# B&R Automation Studio project RS15_RX_30005_r00 (part 6)

### Program Logical/BagMachine_Section/EnvBag/Axis12/A12_Cycle (IEC) - A new program

#### A12_CycleInit.st - Initialization code
```iecst
(********************************************************************
 * COPYRIGHT -- .
 ********************************************************************
 * Program: A12_Cycle
 * File: A12_CycleInit.st
 * Author: dominique
 * Created: November 21, 2011
 ********************************************************************
 * Implementation of program A12_Cycle
 ********************************************************************)

PROGRAM _INIT

  gstCycA[12].CycManTimSet.uiMasterParID := 428 ; // ParID 428 = CTRL Position controller: Input set position (in case real axis)

END_PROGRAM
```

#### A12_Cycle.var - Local variables
```iecst
(********************************************************************
 * COPYRIGHT -- .
 ********************************************************************
 * Program: A12_Cycle
 * File: A12_Cycle.var
 * Author: dominique
 * Created: November 21, 2011
 ********************************************************************
 * Local variables of program A12_Cycle
 ********************************************************************)

VAR
  iTest_          : ARRAY [0..15] OF INT ;
  rTempActPhasDeg : ARRAY[0..15] OF REAL ;
  rTempActOffsetInch : ARRAY[0..15] OF REAL ;
  rTemp_          : ARRAY[0..15] OF REAL ;
  stTON_01        : TON ;
END_VAR

VAR CONSTANT

END_VAR
```

### Program Logical/BagMachine_Section/EnvBag/Axis12/A12_Ref_V1 (IEC) - Reference Routine

#### A12_RefCyclic.ld - Cyclic code
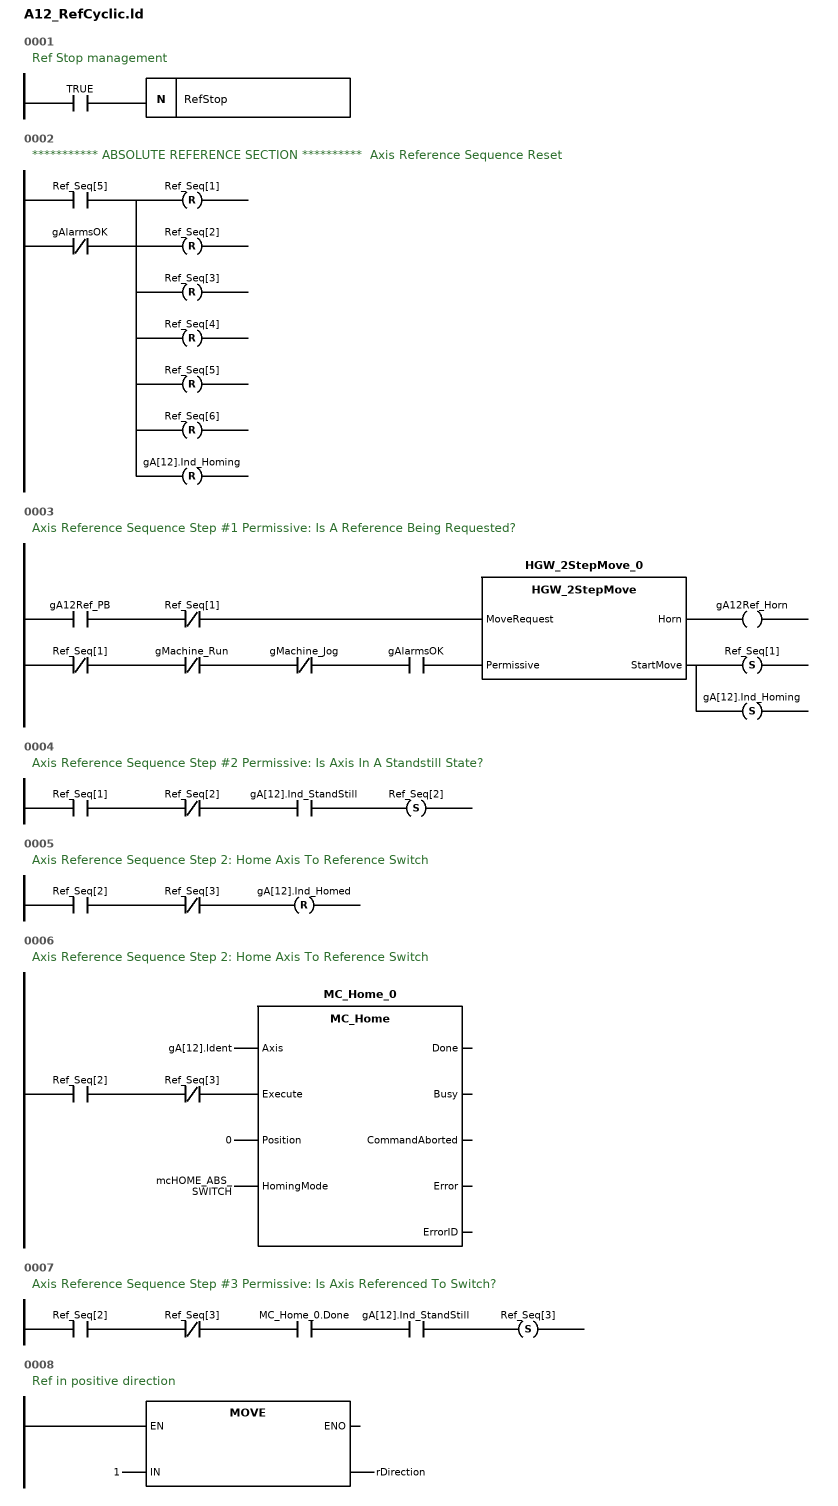
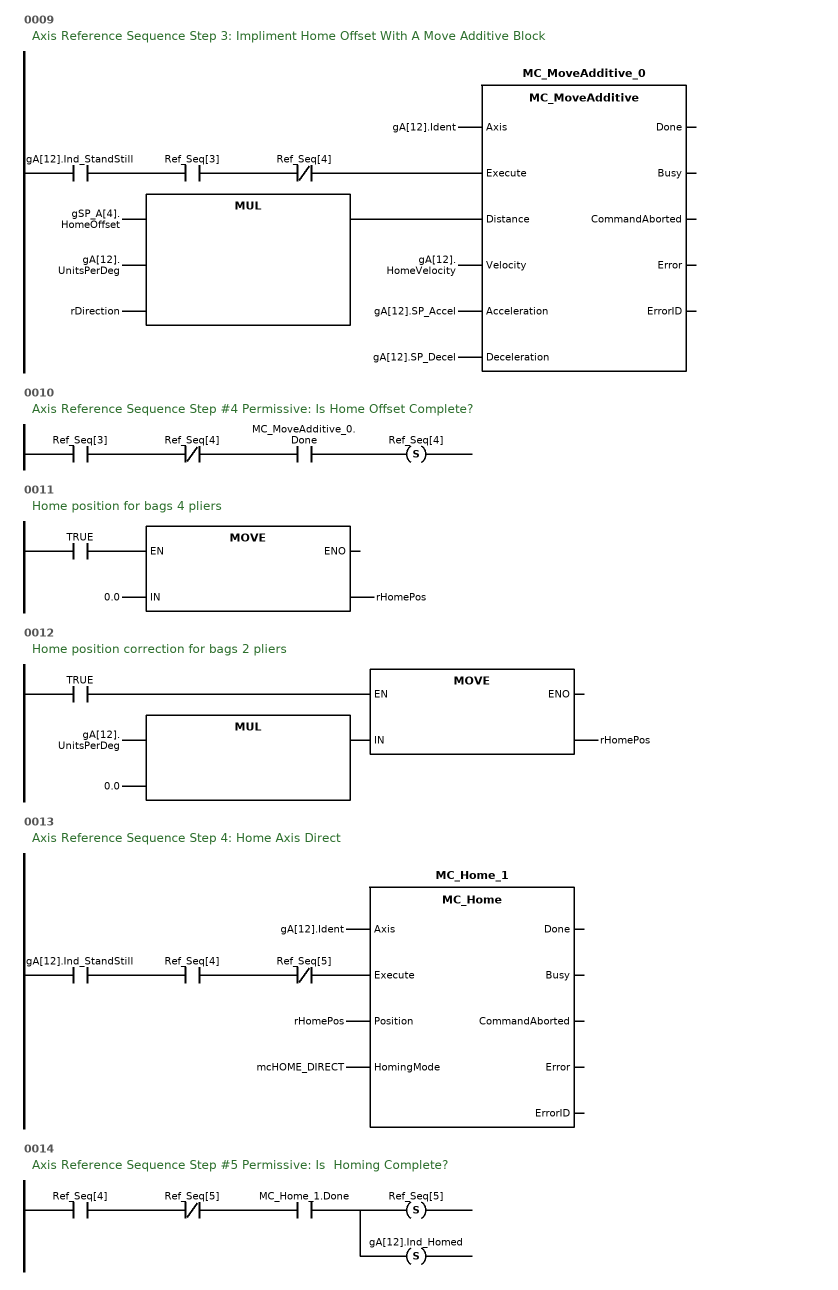
Ladder, written as Structured Text:
```iecst
(********************************************************************
 * COPYRIGHT -- Microsoft
 ********************************************************************
 * Program: A4_Ref
 * File: A4_RefCyclic.ld
 * Author: pkiel
 * Created: July 19, 2011
 ********************************************************************
 * Implementation of program A4_Ref
 ********************************************************************)

PROGRAM _CYCLIC
VAR
    _p1 : BOOL;
    _p2 : BOOL;
END_VAR
(* Network 1: Ref Stop management *)
RefStop;

(* Network 2: *********** ABSOLUTE REFERENCE SECTION **********  Axis Reference Sequence Reset *)
_p1 := Ref_Seq[5];
IF Ref_Seq[5] OR NOT gAlarmsOK THEN Ref_Seq[1] := FALSE; END_IF;
IF _p1 OR NOT gAlarmsOK THEN
    Ref_Seq[2] := FALSE;
    Ref_Seq[3] := FALSE;
    Ref_Seq[4] := FALSE;
    Ref_Seq[5] := FALSE;
    Ref_Seq[6] := FALSE;
    gA[12].Ind_Homing := FALSE;
END_IF;

(* Network 3: Axis Reference Sequence Step #1 Permissive: Is A Reference Being Requested? *)
HGW_2StepMove_0(MoveRequest := gA12Ref_PB AND NOT Ref_Seq[1], Permissive := NOT Ref_Seq[1] AND NOT gMachine_Run AND NOT gMachine_Jog AND gAlarmsOK);
gA12Ref_Horn := HGW_2StepMove_0.Horn;
IF HGW_2StepMove_0.StartMove THEN
    Ref_Seq[1] := TRUE;
    gA[12].Ind_Homing := TRUE;
END_IF;

(* Network 4: Axis Reference Sequence Step #2 Permissive: Is Axis In A Standstill State? *)
IF Ref_Seq[1] AND NOT Ref_Seq[2] AND gA[12].Ind_StandStill THEN Ref_Seq[2] := TRUE; END_IF;

(* Network 5: Axis Reference Sequence Step 2: Home Axis To Reference Switch *)
IF Ref_Seq[2] AND NOT Ref_Seq[3] THEN gA[12].Ind_Homed := FALSE; END_IF;

(* Network 6: Axis Reference Sequence Step 2: Home Axis To Reference Switch *)
MC_Home_0(Axis := gA[12].Ident, Execute := Ref_Seq[2] AND NOT Ref_Seq[3], Position := 0, HomingMode := mcHOME_ABS_SWITCH);

(* Network 7: Axis Reference Sequence Step #3 Permissive: Is Axis Referenced To Switch? *)
IF Ref_Seq[2] AND NOT Ref_Seq[3] AND MC_Home_0.Done AND gA[12].Ind_StandStill THEN
    Ref_Seq[3] := TRUE;
END_IF;

(* Network 8: Ref in positive direction  *)
rDirection := 1;

(* Network 9: Axis Reference Sequence Step 3: Impliment Home Offset With A Move Additive Block *)
MC_MoveAdditive_0(Axis := gA[12].Ident, Execute := gA[12].Ind_StandStill AND Ref_Seq[3] AND NOT Ref_Seq[4], Distance := gSP_A[4].HomeOffset * gA[12].UnitsPerDeg * rDirection, Velocity := gA[12].HomeVelocity, Acceleration := gA[12].SP_Accel, Deceleration := gA[12].SP_Decel);

(* Network 10: Axis Reference Sequence Step #4 Permissive: Is Home Offset Complete? *)
IF Ref_Seq[3] AND NOT Ref_Seq[4] AND MC_MoveAdditive_0.Done THEN Ref_Seq[4] := TRUE; END_IF;

(* Network 11: Home position for bags 4 pliers  *)
rHomePos := 0.0;

(* Network 12: Home position correction for bags 2 pliers *)
rHomePos := gA[12].UnitsPerDeg * 0.0;

(* Network 13: Axis Reference Sequence Step 4: Home Axis Direct *)
MC_Home_1(Axis := gA[12].Ident, Execute := gA[12].Ind_StandStill AND Ref_Seq[4] AND NOT Ref_Seq[5], Position := rHomePos, HomingMode := mcHOME_DIRECT);

(* Network 14: Axis Reference Sequence Step #5 Permissive: Is  Homing Complete? *)
_p2 := Ref_Seq[4] AND NOT Ref_Seq[5] AND MC_Home_1.Done;
IF Ref_Seq[4] AND NOT Ref_Seq[5] AND MC_Home_1.Done THEN Ref_Seq[5] := TRUE; END_IF;
IF _p2 THEN gA[12].Ind_Homed := TRUE; END_IF;
END_PROGRAM
```

### Package Logical/BagMachine_Section/EnvBag/Axis13 - Tearing Envelope Bag Axis     TearEB  Axis

### Program Logical/BagMachine_Section/EnvBag/Axis13/A13_Automat

#### A13_Automat.var
```iecst
(********************************************************************
 * COPYRIGHT -- Microsoft
 ********************************************************************
 * Program: A13_Automat
 * File: A13_Automat.var
 * Author: dominique
 * Created: November 21, 2011
 ********************************************************************
 * Local variables of program A13_Automat
 ********************************************************************)
VAR
	AutData : MC_AUTDATA_TYP;
	AutomatStart : BOOL;
	ErrorID : UINT;
	MasterOffset : REAL;
  MasterParID : UINT;
  uiMasterParID1 : UINT;
  uiSP_MasterParID : UINT;
  uiiSP_Master : UDINT;
  bCmdSynchroOn : BOOL ;
  bCmdSynchroOff : BOOL ;
  bCmdSynchroOn1 : BOOL ;
  bCmdSynchroOff1 : BOOL ;
  uiiSP_MasterFactor : UDINT ;
  uiiSP_SlaveFactor : UDINT ;
	MC_BR_AutControl_0 : MC_BR_AutControl;
  uiMC_BR_AutControl_0_MemoErrorID : UINT ;
  MC_BR_InitMasterParIDTransfer_0 : MC_BR_InitMasterParIDTransfer;
  MC_BR_InitMasterParIDTransfer_1 : MC_BR_InitMasterParIDTransfer;
  ParID_Ready : BOOL;
  ParID_Ready1 : BOOL;
	PositionMOD : DINT;
	PositionOffset : DINT;
	SlaveStartOffset : REAL;
	Synch_Request : BOOL;
  bTest_ : ARRAY[0..9] OF  BOOL;
  iTest_ : ARRAY[0..9] OF  INT;
  rTest_ : ARRAY[0..9] OF  REAL;
  rMaCompDist : REAL ;
  rSPMaPos    : REAL ;
  rOffsetDeg  : REAL ;
  rSlCompDist : REAL ;
  rTemp_      : ARRAY[0..9] OF REAL ;
  usiMemoStat : USINT;
  iIndex : INT ;
  rMaCompDistStat6 : REAL;
  rSlCompDistStat6 : REAL;
  rMasterFactor5 : REAL;
  iiMasterFactor5 : DINT;
  iiSlaveFactor5  : DINT;
  rSlave_AxisPeriod : REAL ;
  rSlave_TimingAxisPeriod : REAL ;
  MC_BR_InitAutState_0 : MC_BR_InitAutState;
  uiInitAutState_0_MemoErrorID : UINT ;
END_VAR
```

#### A13_AutomatCyclic.st
```iecst
(********************************************************************
 * COPYRIGHT -- Microsoft
 ********************************************************************
 * Program: A13_Automat
 * File: A13_AutomatCyclic.st
 * Author: dominique
 * Created: November 21, 2011
 ********************************************************************
 * Implementation of program A13_Automat
 ********************************************************************)

PROGRAM _CYCLIC

    // Synchro ratio Master/Slave
    iIndex := MC_BR_AutControl_0.ActualStateIndex ;
    IF gRecipeActive.bSelEnvBProd THEN
      CASE iIndex OF
        3 : // Master = EnvB Axis
           //gA[13].rRSynNum := 4.0 ;       D.M. 03/02/2012 Pyrollpack_14661 Suppress cause is not correct for offset Virtual Masrter / Slave calculation in A4_Basic and not used in setting mode Automat states 3 and 4
           //gA[13].rRSynDen := 1.0 ;
      ELSE  // Master = Virtual
           gA[13].rRSynNum := 2.0 ;
           gA[13].rRSynDen := 1.0 ;
      END_CASE
    ELSE
      CASE iIndex OF
        3 : // Master = Tearing
           //gA[13].rRSynNum := 4.0 ;
           //gA[13].rRSynDen := 1.0 ;
      ELSE  // Master = Virtual
           IF (g_rNumbPliers <> 0.0) THEN
             gA[13].rRSynNum := 4.0 / g_rNumbPliers ;
           ELSE
             gA[13].rRSynNum := 4.0 ;
           END_IF
           gA[13].rRSynDen := 1.0 ;
      END_CASE
    END_IF

(**** STRAIGHT GEARED CAM AUTOMAT WITH ABSOLUTE PHASE SYNCHRONIZATION FOR ENVELOPE BAG AXIS ***)

(* Set Up Master Position Parameter ID *)

  // Holding+Tearing+EnvBag+TearEB+Drum timing setting
  IF gstCycA[3].CycManTimSet.CmdSynchroOn  OR
     gstCycA[4].CycManTimSet.CmdSynchroOn  OR
     gstCycA[12].CycManTimSet.CmdSynchroOn THEN
    MC_BR_AutControl_0.Signal1 := 1 ;
    MC_BR_AutControl_0.Signal2 := 0 ;
  ELSE
    MC_BR_AutControl_0.Signal1 := 0 ;
    MC_BR_AutControl_0.Signal2 := 1 ;
  END_IF

  // A13 Synchro OK indicator
  gstCycA[3].CycManTimSet.bSynchroOkSlavA[13] := ( MC_BR_InitMasterParIDTransfer_1.Master = gA[12].Ident )                                AND
                                                 ( MC_BR_InitMasterParIDTransfer_1.MasterParID = gstCycA[12].CycManTimSet.uiMasterParID ) AND
                                                 ( MC_BR_AutControl_0.ActualStateIndex = 3 )                                              AND
                                                 gA[13].Ind_SynchronizedMotion AND ParID_Ready ;

  // A13 Synchro OK indicator
  gstCycA[4].CycManTimSet.bSynchroOkSlavA[13] := ( MC_BR_InitMasterParIDTransfer_1.Master = gA[12].Ident )                                AND
                                                 ( MC_BR_InitMasterParIDTransfer_1.MasterParID = gstCycA[12].CycManTimSet.uiMasterParID ) AND
                                                 ( MC_BR_AutControl_0.ActualStateIndex = 3 )                                              AND
                                                 gA[13].Ind_SynchronizedMotion AND ParID_Ready ;

  // A13 Synchro OK indicator
  gstCycA[12].CycManTimSet.bSynchroOkSlavA[13] := ( MC_BR_InitMasterParIDTransfer_1.Master = gA[12].Ident )                                AND
                                                  ( MC_BR_InitMasterParIDTransfer_1.MasterParID = gstCycA[12].CycManTimSet.uiMasterParID ) AND
                                                  ( MC_BR_AutControl_0.ActualStateIndex = 3 )                                              AND
                                                  gA[13].Ind_SynchronizedMotion AND ParID_Ready ;

  // TearEB+Drum timing setting
  IF gstCycA[13].CycManTimSet.bCyc THEN
    IF (gstCycA[13].CycManTimSet.CmdSynchroOn) THEN
      MC_BR_AutControl_0.Signal1 := 0 ;
      MC_BR_AutControl_0.Signal2 := 0 ;
      MC_BR_AutControl_0.Signal3 := 1 ;
    ELSE
      MC_BR_AutControl_0.Signal1 := 0 ;
      MC_BR_AutControl_0.Signal2 := 0 ;
      MC_BR_AutControl_0.Signal3 := 0 ;
    END_IF
  END_IF

  // A13 Synchro OK indicator
  gstCycA[13].CycManTimSet.bSynchroOkSlavA[13] := ( MC_BR_AutControl_0.ActualStateIndex = 2 )   AND
                                                  gA[13].Ind_SynchronizedMotion AND ParID_Ready ;

  IF gstCycA[3].CycManTimSet.bFCyc  AND
     gstCycA[4].CycManTimSet.bFCyc  AND
     gstCycA[12].CycManTimSet.bFCyc AND
     gstCycA[13].CycManTimSet.bFCyc THEN
    MC_BR_AutControl_0.Signal1 := 0 ;
    MC_BR_AutControl_0.Signal2 := 0 ;
    MC_BR_AutControl_0.Signal3 := 0 ;
  END_IF

  // Slave Period
  IF gRecipeActive.bSelEnvBProd THEN
    rSlave_TimingAxisPeriod := gA[13].AxisPeriod * 2.0 ; // EnvB Axis is Master
    rSlave_AxisPeriod       := gA[13].AxisPeriod * 2.0 ; // Virtual Master Axis is Master
  ELSE
    rSlave_TimingAxisPeriod := gA[13].AxisPeriod * 4.0 ; // EnvB Axis is Master
    rSlave_AxisPeriod       := gA[13].AxisPeriod * 4.0 / g_rNumbPliers ; // Virtual Master Axis is Master
  END_IF

  //Synch_Request := gA[13].Cmd_SynchronizedMotion ;
  Synch_Request := gA[13].Cmd_SynchronizedMotion AND NOT(MC_BR_AutControl_0.Stop) ;  // D.M. 26/01/2012 RS26 Pyrollpack_14661 added because it happened that Stop=1 and Synch_Request=1 => MC_BR_AutControl_0 makes fault 29256
  IF (Synch_Request AND NOT ParID_Ready) THEN
    MC_BR_InitMasterParIDTransfer_0.Master:= gA[9].Ident ;
    MC_BR_InitMasterParIDTransfer_0.Slave:=gA[13].Ident;
    MC_BR_InitMasterParIDTransfer_0.MasterParID:= 412 ; // ParID 412 = VAX Position (in case virtual axis)
    MC_BR_InitMasterParIDTransfer_0.SlaveChannel:=0;
    MC_BR_InitMasterParIDTransfer_0.Execute:= 1 ;
    IF (MC_BR_InitMasterParIDTransfer_0.Done) THEN
      MasterParID:=MC_BR_InitMasterParIDTransfer_0.ReceiveParID;
      MC_BR_InitMasterParIDTransfer_0.Execute:=FALSE;
      ParID_Ready1:=1;
    ELSIF (MC_BR_InitMasterParIDTransfer_0.Error) THEN
    (*Store ErrorID in a variable,
      ErrorID is reset on falling edge of 'Execute'*)
      ErrorID:=MC_BR_InitMasterParIDTransfer_0.ErrorID;
      ParID_Ready1:=0;
      MC_BR_InitMasterParIDTransfer_0.Execute:=FALSE;
    END_IF
    MC_BR_InitMasterParIDTransfer_1.Master       := gA[12].Ident ;
    MC_BR_InitMasterParIDTransfer_1.Slave        := gA[13].Ident;
    MC_BR_InitMasterParIDTransfer_1.MasterParID  := gstCycA[13].CycManTimSet.uiMasterParID ;
    MC_BR_InitMasterParIDTransfer_1.SlaveChannel := 3 ;
    MC_BR_InitMasterParIDTransfer_1.Execute      := 1 ;
    IF (MC_BR_InitMasterParIDTransfer_1.Done) AND ParID_Ready1 THEN
      uiMasterParID1:=MC_BR_InitMasterParIDTransfer_1.ReceiveParID;
      MC_BR_InitMasterParIDTransfer_1.Execute:=FALSE;
      ParID_Ready:=1;
    ELSIF (MC_BR_InitMasterParIDTransfer_1.Error) THEN
    (*Store ErrorID in a variable,
      ErrorID is reset on falling edge of 'Execute'*)
      ErrorID:=MC_BR_InitMasterParIDTransfer_1.ErrorID;
      ParID_Ready:=0;
      MC_BR_InitMasterParIDTransfer_1.Execute:=FALSE;
    END_IF
  END_IF
  MC_BR_InitMasterParIDTransfer_0();
  MC_BR_InitMasterParIDTransfer_1();

(**** Initialize Automat Parameters Upon Automat Start Request ****)
  IF (EDGEPOS(ParID_Ready))THEN
    // Master Slave Ratio      Master = Virtual Master Axis
    IF gRecipeActive.bSelEnvBProd THEN
      gA[13].rRSynNum := 2.0 ;
      gA[13].rRSynDen := 1.0 ;
    ELSE
       IF (g_rNumbPliers <> 0.0) THEN
         gA[13].rRSynNum := 4.0 / g_rNumbPliers ;
       ELSE
         gA[13].rRSynNum := 4.0 ;
       END_IF
       gA[13].rRSynDen := 1.0 ;
    END_IF

    //*** Calculate Slave Start Offset ****
      MasterOffset := gRecipeActive.Tearing_Offset+gRecipeActive.Holding_Offset;
      PositionOffset:= REAL_TO_DINT((gA[9].PositionInch-(gA[13].PositionInch-MasterOffset))*1000);
      PositionMOD:= REAL_TO_DINT(gRecipeActive.Repeat*1000);
      SlaveStartOffset:= (DINT_TO_REAL(PositionOffset MOD PositionMOD))/1000;
      IF (SlaveStartOffset >= (0.5*gRecipeActive.Repeat)) THEN
        SlaveStartOffset := SlaveStartOffset - gRecipeActive.Repeat;
      END_IF
      IF (SlaveStartOffset < (-0.5*gRecipeActive.Repeat)) THEN
        SlaveStartOffset := SlaveStartOffset + gRecipeActive.Repeat;
      END_IF

      rSlave_AxisPeriod := gA[13].AxisPeriod * gA[13].rRSynNum/gA[13].rRSynDen ;
      rOffsetDeg := gRecipeActive.rTearEB_PhasMasterDeg ;

      rSPMaPos := (gA[13].PositionDeg - rOffsetDeg)/(gA[13].rRSynNum/gA[13].rRSynDen) ;
      rTemp_[0] := rSPMaPos - gA[9].PositionDeg ;
      rMaCompDist := H_FC_Modulus (
                          IN_rMod := (360 * gA[13].rRSynNum/gA[13].rRSynDen) ,
                          IN_rVar := rTemp_[0]
                                  ) ;

    (*general automat parameter*)
      //AutData.Master            := gA[3].Ident;
      AutData.MasterParID        := MasterParID;
      AutData.StartPosition      := 0;
      AutData.StartInterval      := gA[9].AxisPeriod;
      AutData.MaxMasterVelocity  := gr_rMachMaxSpeed_BPM ;

    //Automat STATE 0 Basis State
      AutData.State[0].Event[0].Type      := ncST_END;
      AutData.State[0].Event[0].Attribute  := ncAT_ONCE;
      IF (rMaCompDist >= 1/gA[9].UnitsPerDeg) AND // rMaCompDist must be >= 1 Units
         gA[13].bSynchroReq                   THEN
        AutData.State[0].Event[0].NextState  := 1;
      ELSE
        rMaCompDist := 1/gA[9].UnitsPerDeg ;
        AutData.State[0].Event[0].NextState := 2;
      END_IF

    //Automat STATE 1 Master/Slave Absolute Phase Correction
      AutData.State[1].MasterParID        := MasterParID;
      AutData.State[1].CamProfileIndex    := 16#FFFF;
      AutData.State[1].MasterFactor       := REAL_TO_UDINT(rMaCompDist * gA[13].UnitsPerDeg) ;
      AutData.State[1].SlaveFactor        := 0 ;
      AutData.State[1].CompMode           := ncOFF;

      AutData.State[1].Event[0].Type      := ncST_END ;
      AutData.State[1].Event[0].Attribute := ncST_END ;
      AutData.State[1].Event[0].NextState := 2 ;

      AutData.State[1].Event[1].Type      := ncSIGNAL1 ;
      AutData.State[1].Event[1].Attribute := ncAT_ONCE ;
      AutData.State[1].Event[1].NextState := 3 ;

      AutData.State[1].Event[2].Type      := ncSIGNAL3 ;
      AutData.State[1].Event[2].Attribute := ncAT_ONCE ;
      AutData.State[1].Event[2].NextState := 2 ;

    //Automat STATE 2 Master/Slave run
      AutData.State[2].MasterParID     := MasterParID;
      AutData.State[2].CamProfileIndex := 16#FFFF;
      AutData.State[2].MasterFactor    := REAL_TO_UDINT(gA[9].AxisPeriod);
      AutData.State[2].SlaveFactor     := REAL_TO_UDINT(rSlave_AxisPeriod);
      AutData.State[2].CompMode        := ncOFF;

      AutData.State[2].Event[0].Type      := ncST_END ;
      AutData.State[2].Event[0].Attribute := ncST_END;
      AutData.State[2].Event[0].NextState := 2;

      AutData.State[2].Event[1].Type      := ncST_END+ncNEGATIVE ;
      AutData.State[2].Event[1].Attribute := ncST_END;
      AutData.State[2].Event[1].NextState := 2;

      AutData.State[2].Event[2].Type      := ncSIGNAL1;
      AutData.State[2].Event[2].Attribute := ncAT_ONCE;
      AutData.State[2].Event[2].NextState := 3;

    //Automat STATE 3 Master/Slave Timing setting
      AutData.State[3].MasterParID     := uiMasterParID1;
      AutData.State[3].CamProfileIndex := 16#FFFF;
      AutData.State[3].MasterFactor    := REAL_TO_UDINT(gA[4].AxisPeriod);
      AutData.State[3].SlaveFactor     := REAL_TO_UDINT(rSlave_TimingAxisPeriod);
      AutData.State[3].CompMode        := ncOFF;

      AutData.State[3].Event[0].Type       := ncST_END ;
      AutData.State[3].Event[0].Attribute  := ncST_END ;
      AutData.State[3].Event[0].NextState  := 3 ;

      AutData.State[3].Event[1].Type       := ncST_END+ncNEGATIVE ;
      AutData.State[3].Event[1].Attribute  := ncST_END ;
      AutData.State[3].Event[1].NextState  := 3 ;

      AutData.State[3].Event[2].Type       := ncSIGNAL2 ;
      AutData.State[3].Event[2].Attribute  := ncAT_ONCE ;
      AutData.State[3].Event[2].NextState  := 2 ;

      MC_BR_AutControl_0.Enable      := 1;
      MC_BR_AutControl_0.AdrAutData  := ADR(AutData);
      MC_BR_AutControl_0.InitAutData := 1;
  END_IF

      (* wait for initialization done or restart *)
      IF ((MC_BR_AutControl_0.AutDataInitialized=1) AND (Synch_Request)) THEN
        MC_BR_AutControl_0.InitAutData := 0;
        MC_BR_AutControl_0.Enable :=1;
        AutomatStart := 1;
        uiMC_BR_AutControl_0_MemoErrorID := 0 ;
      END_IF
      (* check if error occured *)
      IF (MC_BR_AutControl_0.ErrorID <> 0) THEN
        uiMC_BR_AutControl_0_MemoErrorID := MC_BR_AutControl_0.ErrorID ;
        MC_BR_AutControl_0.Enable := 0;
      END_IF

  (******************** ENABLE CAM-AUTOMAT **********************)

  IF (AutomatStart) THEN
      MC_BR_AutControl_0.Start := 1;
      AutomatStart := 0;
  END_IF

  IF (NOT Synch_Request) THEN
      MC_BR_AutControl_0.Stop := 1;
      MC_BR_AutControl_0.Start := 0;
      ParID_Ready := 0;
      ParID_Ready1 := 0;
      IF (MC_BR_AutControl_0.Running=0) THEN
        MC_BR_AutControl_0.Enable := 0;
        MC_BR_AutControl_0.Stop := 0;
        g_bEnvBagSelectChang := 0 ;
      END_IF
   //*************************************************
   // D.M. 26/01/2012 RS26 Pyrollpack_14661 added because after guard fault it happened that Stop=1 and MC_BR_AutControl_0.Enable => not possible to finish MC_BR_AutControl_0 => program locked
      IF MC_BR_AutControl_0.Stop        AND
         NOT(MC_BR_AutControl_0.Enable) THEN
        MC_BR_AutControl_0.Enable := 1 ;
      END_IF
   //*************************************************
  END_IF

  gA[13].Ind_AutomatEnabled:=MC_BR_AutControl_0.Enable;
  gA[13].Ind_CurrentAutomatState:=MC_BR_AutControl_0.ActualStateIndex;
  gA[13].Ind_bSynchroOK := (MC_BR_AutControl_0.ActualStateIndex >= 2) AND gA[13].Ind_SynchronizedMotion ; ;

  (********************** MC_AUTCONTROL *************************)
  MC_BR_AutControl_0.Slave:= gA[13].Ident;
  MC_BR_AutControl_0();

(******************** UPDATE CAM-AUTOMAT STATE 2 **********************)
  IF g_bEnvBagSelectChang                      AND
     (MC_BR_AutControl_0.ActualStateIndex = 2) THEN
    MC_BR_InitAutState_0.Execute := 1 ;
    uiInitAutState_0_MemoErrorID := 0 ;
  END_IF
  MC_BR_InitAutState_0.MasterParID     := MasterParID ;
  MC_BR_InitAutState_0.Slave           := gA[13].Ident ;
  MC_BR_InitAutState_0.StateIndex      := 2 ;
  MC_BR_InitAutState_0.CamProfileIndex := 16#FFFF ;
  MC_BR_InitAutState_0.MasterFactor    := REAL_TO_UDINT(gA[9].AxisPeriod) ;
  MC_BR_InitAutState_0.SlaveFactor     := REAL_TO_DINT(rSlave_AxisPeriod) ;
  MC_BR_InitAutState_0.CompMode        := ncOFF ;
  MC_BR_InitAutState_0() ;

  IF (MC_BR_InitAutState_0.Done)  OR
     (MC_BR_InitAutState_0.Error) THEN
    MC_BR_InitAutState_0.Execute := 0;
    uiInitAutState_0_MemoErrorID := MC_BR_InitAutState_0.ErrorID ;
  END_IF

END_PROGRAM
```

### Program Logical/BagMachine_Section/EnvBag/Axis13/A13_Basic (IEC)

#### A13_BasicInit.st - Initialization code
```iecst
(********************************************************************
 * COPYRIGHT -- Microsoft
 ********************************************************************
 * Program: A13_Basic
 * File: A13_BasicInit.st
 * Author: dominique
 * Created: November 21, 2011
 ********************************************************************
 * Implementation of program A13_Basic
 ********************************************************************)

PROGRAM _INIT

	(* Axis Setpoint Variables *)
		gA[13].SP_MotorPPR := 36000 * 2 / 7 ;
		gA[13].SP_GearBoxInput:= 7;
		gA[13].SP_GearBoxOutput:= 2;
		gA[13].AxisPeriod := 36000 ; // because of limited precsision  (gA[13].SP_MotorPPR*gA[13].SP_GearBoxInput/gA[13].SP_GearBoxOutput) = 35997.5 insted of 36000 and then the synchro is not correct
		gA[13].UnitsPerDeg := gA[13].AxisPeriod/360;
		gA[13].SP_Accel := 0.2*gA[13].AxisPeriod;
		gA[13].SP_Decel := 0.4*gA[13].AxisPeriod;
		gA[13].SP_EStopDecel := 1000.0*gA[13].AxisPeriod; // Stop axis from 1000 tr/min in 1s
		gA[13].HomeVelocity := 6*gA[13].AxisPeriod/60;
    gA[13].rSP_CorPosVel := 0.0 ;
    gA[13].rSP_OverrideV := 1.0 ;
    gA[13].rSP_OverrideA := 1.0 ;
    gA[13].Cmd_EStopDisable := 0 ;

	(* access master axis *)
		AxisErrorNcAccess := ncaccess(ncACP10MAN, ADR('Axis13'), ADR(gA[13].Ident));

	(* Trigger Initialization Of ModPosition *)
		InitModPosition:=1;

END_PROGRAM
```

### Program Logical/BagMachine_Section/EnvBag/Axis13/A13_Control (IEC)

#### A13_ControlCyclic.ld - Cyclic code
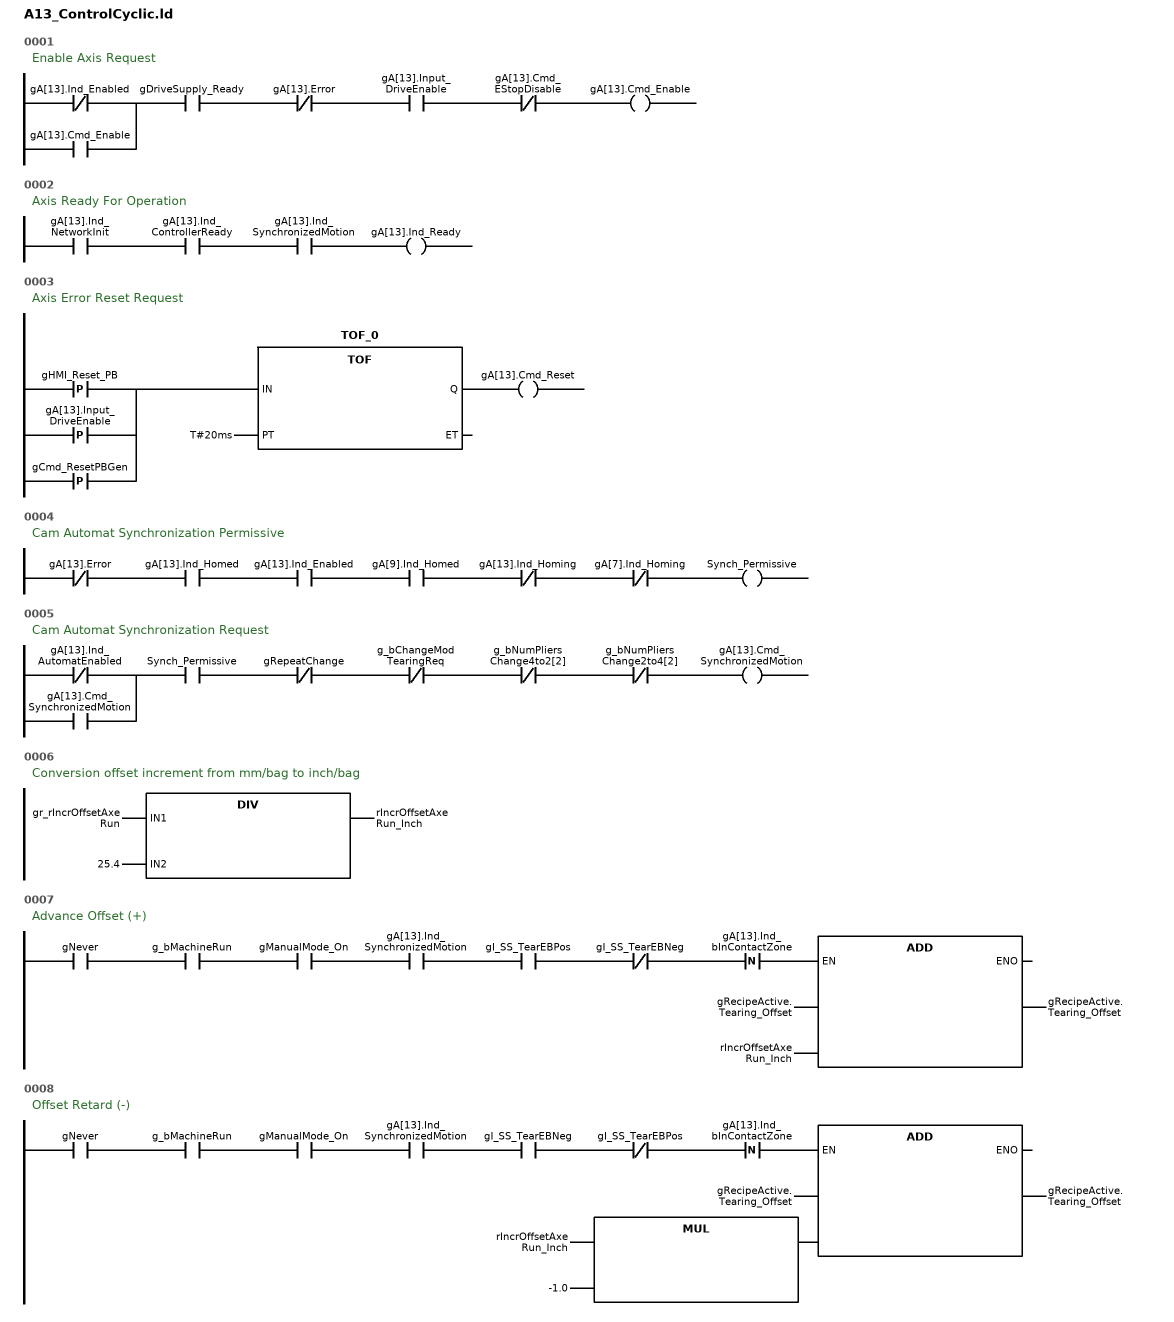
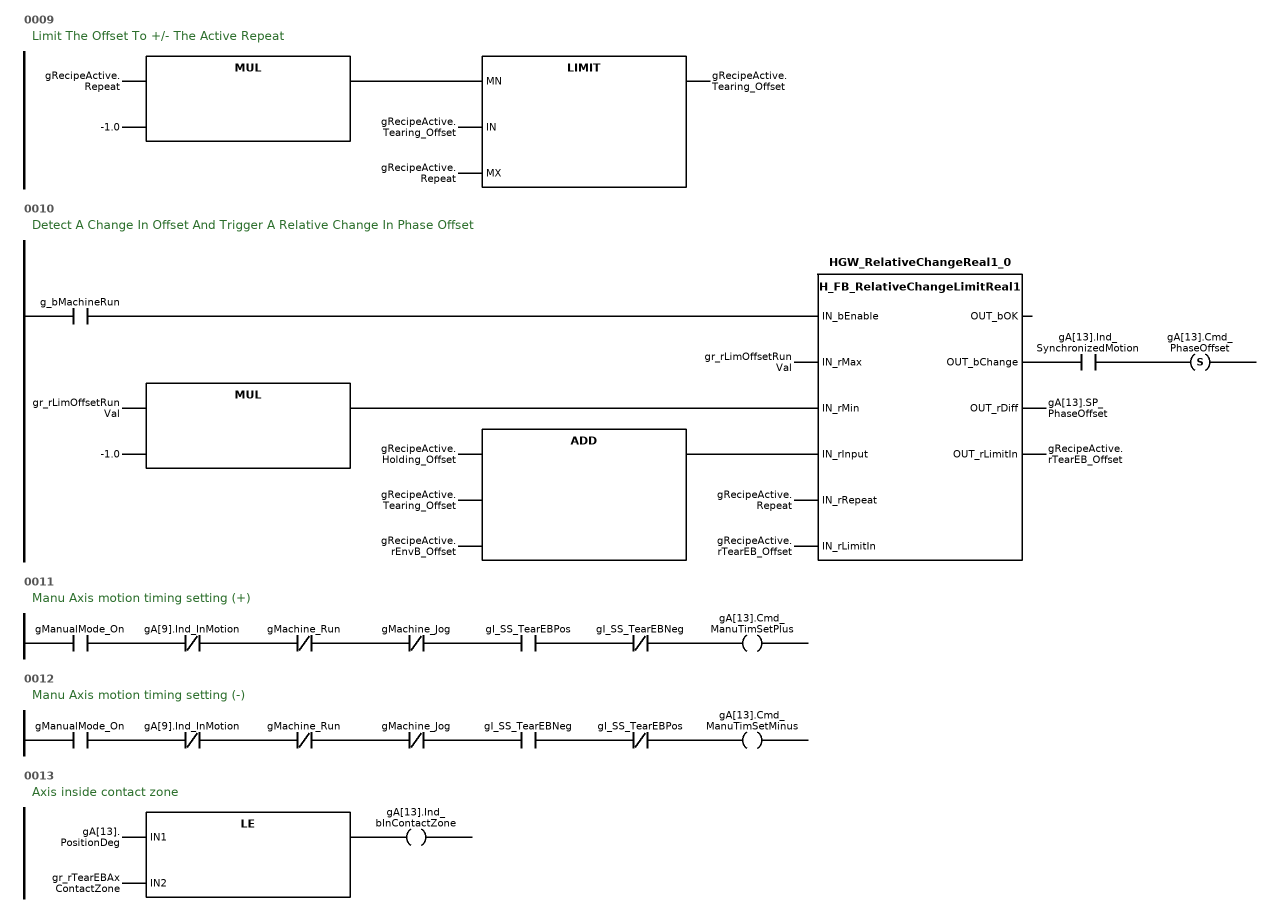
Ladder, written as Structured Text:
```iecst
(********************************************************************
 * COPYRIGHT -- Microsoft
 ********************************************************************
 * Program: A4_Control
 * File: A4_ControlCyclic.ld
 * Author: pkiel
 * Created: July 13, 2011
 ********************************************************************
 * Implementation of program A4_Control
 ********************************************************************)

PROGRAM _CYCLIC
VAR
    _e1 : R_TRIG;
    _e2 : R_TRIG;
    _e3 : R_TRIG;
    _e4 : F_TRIG;
    _e5 : F_TRIG;
END_VAR
(* Network 1: Enable Axis Request *)
gA[13].Cmd_Enable := (NOT gA[13].Ind_Enabled OR gA[13].Cmd_Enable) AND gDriveSupply_Ready AND NOT gA[13].Error AND gA[13].Input_DriveEnable AND NOT gA[13].Cmd_EStopDisable;

(* Network 2: Axis Ready For Operation *)
gA[13].Ind_Ready := gA[13].Ind_NetworkInit AND gA[13].Ind_ControllerReady AND gA[13].Ind_SynchronizedMotion;

(* Network 3: Axis Error Reset Request *)
_e1(CLK := gHMI_Reset_PB);
_e2(CLK := gA[13].Input_DriveEnable);
_e3(CLK := gCmd_ResetPBGen);
TOF_0(IN := _e1.Q OR _e2.Q OR _e3.Q, PT := T#20ms);
gA[13].Cmd_Reset := TOF_0.Q;

(* Network 4: Cam Automat Synchronization Permissive *)
Synch_Permissive := NOT gA[13].Error AND gA[13].Ind_Homed AND gA[13].Ind_Enabled AND gA[9].Ind_Homed AND NOT gA[13].Ind_Homing AND NOT gA[7].Ind_Homing;

(* Network 5: Cam Automat Synchronization Request *)
gA[13].Cmd_SynchronizedMotion := (NOT gA[13].Ind_AutomatEnabled OR gA[13].Cmd_SynchronizedMotion) AND Synch_Permissive AND NOT gRepeatChange AND NOT g_bChangeModTearingReq AND NOT g_bNumPliersChange4to2[2] AND NOT g_bNumPliersChange2to4[2];

(* Network 6: Conversion offset increment from mm/bag to inch/bag *)
rIncrOffsetAxeRun_Inch := gr_rIncrOffsetAxeRun / 25.4;

(* Network 7: Advance Offset (+) *)
_e4(CLK := gA[13].Ind_bInContactZone);
IF gNever AND g_bMachineRun AND gManualMode_On AND gA[13].Ind_SynchronizedMotion AND gI_SS_TearEBPos AND NOT gI_SS_TearEBNeg AND _e4.Q THEN
    gRecipeActive.Tearing_Offset := gRecipeActive.Tearing_Offset + rIncrOffsetAxeRun_Inch;
END_IF;

(* Network 8: Offset Retard (-) *)
_e5(CLK := gA[13].Ind_bInContactZone);
IF gNever AND g_bMachineRun AND gManualMode_On AND gA[13].Ind_SynchronizedMotion AND gI_SS_TearEBNeg AND NOT gI_SS_TearEBPos AND _e5.Q THEN
    gRecipeActive.Tearing_Offset := gRecipeActive.Tearing_Offset + (rIncrOffsetAxeRun_Inch * -1.0);
END_IF;

(* Network 9: Limit The Offset To +/- The Active Repeat *)
gRecipeActive.Tearing_Offset := LIMIT(MN := gRecipeActive.Repeat * -1.0, IN := gRecipeActive.Tearing_Offset, MX := gRecipeActive.Repeat);

(* Network 10: Detect A Change In Offset And Trigger A Relative Change In Phase Offset *)
HGW_RelativeChangeReal1_0(IN_bEnable := g_bMachineRun, IN_rMax := gr_rLimOffsetRunVal, IN_rMin := gr_rLimOffsetRunVal * -1.0, IN_rInput := gRecipeActive.Holding_Offset + gRecipeActive.Tearing_Offset + gRecipeActive.rEnvB_Offset, IN_rRepeat := gRecipeActive.Repeat, IN_rLimitIn := gRecipeActive.rTearEB_Offset);
IF HGW_RelativeChangeReal1_0.OUT_bChange AND gA[13].Ind_SynchronizedMotion THEN
    gA[13].Cmd_PhaseOffset := TRUE;
END_IF;
gA[13].SP_PhaseOffset := HGW_RelativeChangeReal1_0.OUT_rDiff;
gRecipeActive.rTearEB_Offset := HGW_RelativeChangeReal1_0.OUT_rLimitIn;

(* Network 11: Manu Axis motion timing setting (+) *)
gA[13].Cmd_ManuTimSetPlus := gManualMode_On AND NOT gA[9].Ind_InMotion AND NOT gMachine_Run AND NOT gMachine_Jog AND gI_SS_TearEBPos AND NOT gI_SS_TearEBNeg;

(* Network 12: Manu Axis motion timing setting (-) *)
gA[13].Cmd_ManuTimSetMinus := gManualMode_On AND NOT gA[9].Ind_InMotion AND NOT gMachine_Run AND NOT gMachine_Jog AND gI_SS_TearEBNeg AND NOT gI_SS_TearEBPos;

(* Network 13: Axis inside contact zone *)
gA[13].Ind_bInContactZone := gA[13].PositionDeg <= gr_rTearEBAxContactZone;
END_PROGRAM
```

### Program Logical/BagMachine_Section/EnvBag/Axis13/A13_Cycle (IEC)

#### A13_CycleCyclic.st - Cyclic code
```iecst
(********************************************************************
 * COPYRIGHT -- .
 ********************************************************************
 * Program: A13_Cycle
 * File: A13_CycleCyclic.st
 * Author: dominique
 * Created: November 21, 2011
 ********************************************************************
 * Implementation of program A13_Cycle
 ********************************************************************)

PROGRAM _CYCLIC

// Manu axis movement for timing setting

    //---------------------------------------------------------------------------------------------------------------------
    // Tearing timing setting cycle
    //---------------------------------------------------------------------------------------------------------------------
    // Start cycle
    gstCycA[13].CycManTimSet.CmdStart := ( gA[13].Cmd_ManuTimSetPlus        OR
                                           gA[13].Cmd_ManuTimSetMinus )     AND
                                         ( NOT(g_bCycManTimeSetOn)          OR
                                           gstCycA[13].CycManTimSet.bSCyc ) AND
                                         gA[13].Ind_Ready                   AND
                                         gA[7].Ind_Ready                    ;
    IF gstCycA[13].CycManTimSet.CmdStart THEN
      gstCycA[13].CycManTimSet.bSCyc := 1 ;
    END_IF ;

    //----------------------------------------------------------------------
    // Cycle at rest
    IF NOT(gstCycA[13].CycManTimSet.bSCyc) AND
       1                                 THEN
      IF NOT( gstCycA[13].CycManTimSet.bFCyc ) THEN
        // Init after cycle unpropaly ended
        gstCycA[13].CycManTimSet.bFCyc := 1 ;
        gstCycA[13].CycManTimSet.bCyc  := 0 ;

        gstCycA[13].CycManTimSet.CmdMov       := 0 ;
        gstCycA[13].CycManTimSet.CmdStop      := 0 ;
        gstCycA[13].CycManTimSet.CmdSynchroOn := 0 ;
      END_IF
      gstCycA[13].CycManTimSet.iStep := 0 ;
      RETURN ;
    ELSE
    //----------------------------------------------------------------------
    // Cycle running

      // Permanent conditions
      IF NOT(gA[13].Ind_Ready)                  OR
         NOT(gA[7].Ind_Ready)                  OR
         NOT(gstCycA[13].CycManTimSet.CmdStart) AND
         (gstCycA[13].CycManTimSet.iStep <= 2)  THEN
        gstCycA[13].CycManTimSet.bSCyc := 0 ;
        RETURN ;
      END_IF

      // Permanent actions
      stTON_01 (
            IN := ( gstCycA[13].CycManTimSet.iStep = C_iSTEP_0 ) ,
            PT := T#30ms
               ) ;

    END_IF
    //----------------------------------------------------------------------
    // Cycle steps

        CASE gstCycA[13].CycManTimSet.iStep OF

        C_iSTEP_0 :
         //----------------------------------------------
         // Etape 1 : Initialisation
         //----------------------------------------------
          IF stTON_01.Q THEN
            gstCycA[13].CycManTimSet.iStep := C_iSTEP_1 ;

            // Action Step 1
            gstCycA[13].CycManTimSet.bFCyc := 0 ;
            gstCycA[13].CycManTimSet.bCyc  := 1 ;
          END_IF

        C_iSTEP_1 :
         //----------------------------------------------
         // Etape 2 : Synchro Drum on Tearing
         //----------------------------------------------
          IF TRUE THEN
            gstCycA[13].CycManTimSet.iStep := C_iSTEP_2 ;

            // Action Step 2
            gstCycA[13].CycManTimSet.CmdSynchroOn := 1 ;
          END_IF

        C_iSTEP_2 :
         //----------------------------------------------
         // Step 3 : Activation motion and Stop waiting
         //----------------------------------------------
          IF gstCycA[13].CycManTimSet.bSynchroOkSlavA[7]  AND
             gstCycA[13].CycManTimSet.bSynchroOkSlavA[13] THEN
            gstCycA[13].CycManTimSet.iStep := C_iSTEP_3 ;

            // Action Step 3
            gstCycA[13].CycManTimSet.CmdMov  := 1 ;
            gstCycA[13].CycManTimSet.CmdStop := 0 ;
            // Stop waiting
          END_IF

        C_iSTEP_3 :
         //----------------------------------------------
         // Step 4 : Stop motion and End stop waiting
         //----------------------------------------------
          IF NOT(gstCycA[13].CycManTimSet.CmdStart) THEN
            gstCycA[13].CycManTimSet.iStep := C_iSTEP_4 ;

            // Action Step 4
            gstCycA[13].CycManTimSet.CmdMov  := 0 ;
            gstCycA[13].CycManTimSet.CmdStop := 1 ;
            // End stop waiting
          END_IF

        C_iSTEP_4 :
         //----------------------------------------------
         // Step 3 : Activation motion and Stop waiting
         // Step 5 : Cut synchro
         //----------------------------------------------
          // Condition Step3
          IF gstCycA[13].CycManTimSet.CmdStart THEN
            gstCycA[13].CycManTimSet.iStep := C_iSTEP_3 ;

            // Action Step 3
            gstCycA[13].CycManTimSet.CmdMov  := 1 ;
            gstCycA[13].CycManTimSet.CmdStop := 0 ;
            // Stop waiting
            RETURN ;
          END_IF ;
          // Condition Step5
          IF NOT(gstCycA[13].CycManTimSet.CmdStop) THEN
            gstCycA[13].CycManTimSet.iStep := C_iSTEP_5 ;

            // Action Step 5
            gstCycA[13].CycManTimSet.CmdSynchroOn := 0 ;
          END_IF

        C_iSTEP_5 :
         //----------------------------------------------
         // Step 6 : New offset calculation
         //----------------------------------------------
          IF NOT(gstCycA[13].CycManTimSet.bSynchroOkSlavA[7]) THEN
            gstCycA[13].CycManTimSet.iStep := C_iSTEP_6 ;

            // Action Step 6
            // Memo Actual phase Offset
            rTempActPhasDeg[13]    := gRecipeActive.rTearEB_PhasMasterDeg;
            rTempActOffsetInch[13] := gRecipeActive.rTearEB_Offset ;
            // Update phase
            gRecipeActive.rDrum_PhasMasterDeg   := gA[7].rActPhasDeg ;
            gRecipeActive.rTearEB_PhasMasterDeg := gA[13].rActPhasDeg ;
            // Update Offset
            rTemp_[13] := rTempActOffsetInch[13] + (gRecipeActive.rTearEB_PhasMasterDeg - rTempActPhasDeg[13])/(gA[13].rRSynNum/gA[13].rRSynDen)*gA[13].InchPerDeg ;
            gRecipeActive.rTearEB_Offset := H_FC_Modulus (IN_rMod := gRecipeActive.Repeat, IN_rVar := rTemp_[13]) ;
          END_IF

        C_iSTEP_6 :
         //----------------------------------------------
         // Step 0 : First step
         //----------------------------------------------
          IF NOT(gstCycA[13].CycManTimSet.bSynchroOkSlavA[7]) AND
             (gA[13].Ind_CurrentAutomatState <> 3)            THEN
            gstCycA[13].CycManTimSet.iStep := C_iSTEP_0 ;

            // Action Step 0
            gstCycA[13].CycManTimSet.bSCyc := 0 ;
            gstCycA[13].CycManTimSet.bFCyc := 1 ;
            gstCycA[13].CycManTimSet.bCyc  := 0 ;
          END_IF
        END_CASE
    //---------------------------------------------------------------------------------------------------------------------

END_PROGRAM
```

#### A13_CycleInit.st - Initialization code
```iecst
(********************************************************************
 * COPYRIGHT -- .
 ********************************************************************
 * Program: A13_Cycle
 * File: A13_CycleInit.st
 * Author: dominique
 * Created: November 21, 2011
 ********************************************************************
 * Implementation of program A13_Cycle
 ********************************************************************)

PROGRAM _INIT

  gstCycA[13].CycManTimSet.uiMasterParID := 428 ; // ParID 428 = CTRL Position controller: Input set position (in case real axis)

END_PROGRAM
```

#### A13_Cycle.var - Local variables
```iecst
(********************************************************************
 * COPYRIGHT -- .
 ********************************************************************
 * Program: A13_Cycle
 * File: A13_Cycle.var
 * Author: dominique
 * Created: November 21, 2011
 ********************************************************************
 * Local variables of program A13_Cycle
 ********************************************************************)

VAR
  iTest_          : ARRAY [0..15] OF INT ;
  rTempActPhasDeg : ARRAY[0..15] OF REAL ;
  rTempActOffsetInch : ARRAY[0..15] OF REAL ;
  rTemp_          : ARRAY[0..15] OF REAL ;
  stTON_01        : TON ;
END_VAR

VAR CONSTANT

END_VAR
```

- Data object Logical/BagMachine_Section/EnvBag/Axis13/A13_Init (Ax) (no source held here)

- Data object Logical/BagMachine_Section/EnvBag/Axis13/A13_Par (Apt) (no source held here)

### A13_Ref.var
```iecst
(********************************************************************
 * COPYRIGHT -- Microsoft
 ********************************************************************
 * Program: A13_Ref
 * File: A13_Ref.var
 * Author: dominique
 * Created: November 21, 2011
 ********************************************************************
 * Local variables of program A13_Ref
 ********************************************************************)
VAR
	HGW_2StepMove_0 : HGW_2StepMove;
	MC_Home_0 : MC_Home;
	MC_Home_1 : MC_Home;
	MC_MoveAdditive_0 : MC_MoveAdditive;
	Ref_Seq : ARRAY[0..10] OF BOOL;

  rHomePos   : REAL ;
  rDirection : REAL ;
END_VAR
```

### Package Logical/BagMachine_Section/HotMicroPerf - Axis

### Program Logical/BagMachine_Section/HotMicroPerf/HMPerf_Gen (IEC) - General Hot Micro Perf control

#### HMPerf_GenCyclic.st - Cyclic code
```iecst
(********************************************************************
 * COPYRIGHT -- .
 ********************************************************************
 * Program: HMPerf_Gen
 * File: HMPerf_GenCyclic.st
 * Author: dominique
 * Created: November 05, 2011
 ********************************************************************
 * Implementation of program HMPerf_Gen
 ********************************************************************)

PROGRAM _CYCLIC
  // ----------------------------------------------------------------------------------
  // Status
  bReadyInd := gA[15].Ind_Ready ;

  // Hot Micro Perf Light On
  gQ_HMP_LightOn := g_stHMPerfCyc.bCyc ;

  // ----------------------------------------------------------------------------------
  // Operation mode Hot Micro Perf
  // Cas On
  bOnReq := gI_HMP_On_PB AND gI_HMP_Off_PB AND NOT(g_stHMPerfCyc.bSelProd) ;
  IF bOnReq THEN
    IF NOT(gA[9].Ind_InMotion) AND
       gA[15].Ind_Ready        AND
       NOT(g_bIndEStop)        AND
       1                       THEN
      g_stHMPerfCyc.bSelProd := 1 ;
    ELSE
      g_stHMPerfCyc.bSelProd := 0 ;
      gI_HMP_On_PB := 0 ;
    END_IF ;
  END_IF ;

  // Cas Off
  bOffReq := NOT(gI_HMP_Off_PB) AND g_stHMPerfCyc.bSelProd ;
  IF bOffReq THEN
    IF 1                       AND
       //NOT(gA[9].Ind_InMotion) AND
       1                       THEN
      g_stHMPerfCyc.bStopReq := 1 ;
    ELSE
      g_stHMPerfCyc.bStopReq := 0 ;
      gI_HMP_On_PB := 1 ;
    END_IF ;
  END_IF ;

  // ----------------------------------------------------------------------------------
  // Operation mode Hot Micro Perf
  // Cas Interrupt
  bInterruptReq := HMI_HMPerf_bModePB AND NOT(gRecipeActive.bHMPerf_Mode) ;
  IF bInterruptReq THEN
    IF NOT(gA[9].Ind_InMotion) AND
       1                       THEN
      gRecipeActive.bHMPerf_Mode:= 1 ;
    ELSE
      gRecipeActive.bHMPerf_Mode := 0 ;
    END_IF ;
  END_IF ;

  // Cas Continu
  bContinuReq := NOT(HMI_HMPerf_bModePB) AND gRecipeActive.bHMPerf_Mode ;
  IF bContinuReq THEN
    IF 1                       AND
       NOT(gA[9].Ind_InMotion) AND
       1                       THEN
      gRecipeActive.bHMPerf_Mode := 0 ;
    ELSE
      gRecipeActive.bHMPerf_Mode := 1 ;
    END_IF
  END_IF

  // ----------------------------------------------------------------------------------
  // Axis ativation
  gA[15].bActive := g_stHMPerfCyc.bSelProd ;

  // ----------------------------------------------------------------------------------
  // Operator tool size set point Limit
  gRecipeActive.rHotMicroPerfSize_in := LIMIT(g_rMinBagSize_Inch,gRecipeActive.rHotMicroPerfSize_in,g_rMaxBagSize_Inch) ;

  // ----------------------------------------------------------------------------------
  // Tool size change lock
  bToolSizeLock := gRecipeActive.bHMPerf_Mode OR
                   g_bMachineRun              ;

  // Up Visible and Lock
  IF gRecipeActive.bHMPerf_Mode THEN
    iToolUpVisibl := 0 ;
   ELSE
    iToolUpVisibl := 1 ;
  END_IF
  bToolUpLock := g_bMachineRun ;

  gRecipeActive.iHMPerf_Up := LIMIT(1,gRecipeActive.iHMPerf_Up,4) ;
  IF gRecipeActive.bHMPerf_Mode THEN
    gRecipeActive.rHotMicroPerfSize_in := gRecipeActive.Repeat * gRecipeActive.iHMPerf_Up ;
  END_IF ;

  // Offset Lock
  bOffsetLock := 0 ; //NOT(g_stHMPerfCyc.bSynchro_OK) ;

  // ----------------------------------------------------------------------------------
  // Operation State
  IF g_stHMPerfCyc.bSlowRot_OK THEN  // Slow Rotation
    iOperState := 1 ;
    uiOperStateCol_Ind := gViolet_5 + + gWhite * 256 ;
  END_IF ;

  IF g_stHMPerfCyc.bSynchro_OK THEN  // Sychronized
    iOperState := 2 ;
    uiOperStateCol_Ind := gGreen + gBlack * 256 ;
  END_IF ;

  IF g_stHMPerfCyc.bFaultCond THEN  // Fault
    iOperState := 3 ;
    uiOperStateCol_Ind := gRed + gBlack * 256 ;
  END_IF ;

  IF NOT(g_stHMPerfCyc.bCyc) THEN  // Off
    iOperState := 0 ;
    uiOperStateCol_Ind := gBlue + gWhite * 256 ;
  END_IF ;

  // ----------------------------------------------------------------------------------
  // Heater State
  IF gQ_HMP_Heater THEN  // On
    iHeatState := 1 ;
    uiHeatStateCol_Ind := gGreen + gBlack * 256 ;
  END_IF ;

  IF NOT(gQ_HMP_Heater) THEN  // Off
    iHeatState := 0 ;
    uiHeatStateCol_Ind := gBlue + gWhite * 256 ;
  END_IF ;

END_PROGRAM
```

- Data object Logical/BagMachine_Section/HotMicroPerf/Axis15/A15_Par (Apt) - Servo Axis Parameter File (no source held here)

### Program Logical/BagMachine_Section/HotMicroPerf/Axis15/A15_Basic (IEC) - Basic Servo

#### A15_Basic.var
```iecst
(********************************************************************
 * COPYRIGHT -- Microsoft
 ********************************************************************
 * Program: A15_Basic
 * File: A15_Basic.var
 * Author: dominique
 * Created: November 03, 2011
 ********************************************************************
 * Local variables of program A15_Basic
 ********************************************************************)
VAR
	AutoAck : BOOL;
	AxisErrorNcAccess : UINT;
	DriveStatus : MC_DRIVESTATUS_TYP;
	HomeRestore : BOOL;
	InitEndlessPosition : BOOL;
	InitModPos_Done : BOOL;
	InitModPosition : BOOL;
	MC_BR_InitEndlessPosition_0 : MC_BR_InitEndlessPosition;
	MC_BR_InitModPos_0 : MC_BR_InitModPos;
  uiInitModPos0_ErrorID : UINT ;
  MC_BR_Phasing_0 : MC_BR_Phasing;
  rSP_PhaseOffset  : REAL ;
  rSP_ShiftVal     : REAL ;
  rShiftSign       : REAL ;
  rMaxShift        : REAL ;
  bCmd_PhaseOffset : BOOL ;
  MC_BR_Phasing_1 : MC_BR_Phasing;
	MC_BR_ReadDriveStatus_0 : MC_BR_ReadDriveStatus;
	MC_Home_0 : MC_Home;
	MC_Home_1 : MC_Home;
	MC_MoveVelocity_0 : MC_MoveVelocity;
	MC_Power_0 : MC_Power;
	MC_ReadActualPosition_0 : MC_ReadActualPosition;
	MC_ReadActualTorque_0 : MC_ReadActualTorque;
	MC_ReadActualVelocity_0 : MC_ReadActualVelocity;
	MC_ReadAxisError_0 : MC_ReadAxisError;
	MC_ReadStatus_0 : MC_ReadStatus;
	MC_Reset_0 : MC_Reset;
  MC_Stop_0 : MC_Stop;
  MC_Stop_1 : MC_Stop;
  MC_Halt_0 : MC_Halt;
	ResetError : BOOL;
  rTemp_ : ARRAY[0..9] OF REAL ;
  bTest_ : ARRAY[0..9] OF BOOL ;
  rTest_ : ARRAY[0..9] OF REAL ;
  iTest_ : ARRAY[0..9] OF INT ;
  rAxisTimSet_SP_Vel  : REAL ; (*Set point Velocity for Axis manual timing setting cycle, in units/s*)
  rAxisTimSet_SP_Acc  : REAL ; (*Set point Acceleration for Axis manual timing setting cycle, in units/s²*)
  rAxisTimSet_SP_Dec  : REAL ; (*Set point Deceleration for Axis manual timing setting cycle, in units/s²*)
  uiAxisTimSet_SP_Dir : USINT ; (*Set point Direction for Axis manual timing setting cycle*)
  uiAxisTimSet_SP_ShiftAppMode : UINT ; (*Set point Shit Application mode for phasing Axis manual timing setting cycle*)
  rTempActPhasDeg : REAL;
  rA9PosCorDeg  : REAL;
  rRepeatMetric : REAL;
  MC_SetOverride_0 : MC_SetOverride;

  iiSP_SlPos_U  : DINT ; (*On Slave side, input set point position of the position controller ParID 428, in unit*)
  rSP_SlPos_Deg : REAL ; (*On Slave side, input set point position of the position controller ParID 428, in deg*)
  iiSP_MaPos_U  : DINT ; (*On Master side, input set point position of the position controller ParID 412, in unit*)
  rSP_MaPos_Deg : REAL ; (*On Master side, input set point position of the position controller ParID 412, in deg*)
  MC_BR_CyclicRead_0 : MC_BR_CyclicRead ;
  MC_BR_CyclicRead_1 : MC_BR_CyclicRead ;

  bChangeModReq : BOOL ;
  uiOffsetStat  : UINT ;
  st_TON_0 : TON ;
END_VAR
```

#### A15_BasicCyclic.st
```iecst
(********************************************************************
 * COPYRIGHT -- Microsoft
 ********************************************************************
 * Program: A15_Basic
 * File: A15_BasicCyclic.st
 * Author: dominique
 * Created: November 03, 2011
 ********************************************************************
 * Implementation of program A15_Basic
 ********************************************************************)

PROGRAM _CYCLIC

	gA[15].UnitsPerInch := gA[15].AxisPeriod/gRecipeActive.Repeat;
  gA[15].InchPerDeg := gA[15].UnitsPerDeg / gA[15].UnitsPerInch ;
  gA[15].rRSynNum := 1 ;
  gA[15].rRSynDen := gRecipeActive.iHMPerf_Up ;

	IF (gA[15].Ident<>0) THEN

	//*********************** READ DRIVE STATUS ************************
	(* Access to the following bools:
	gA[x]_DriveStatus.Simulation			: If TRUE, simulation mode is active
	gA[x]_DriveStatus.NetworkInit			: If TRUE, the network is initialized
	gA[x]_DriveStatus.HomeSwitch			: If TRUE, the digital reference switch input is active
	gA[x]_DriveStatus.PosHWSwitch			: If TRUE, the positive hardware end switch is active
	gA[x]_DriveStatus.NegHWSwitch			: If TRUE, the negative hardware end switch is active
	gA[x]_DriveStatus.Trigger1				: If TRUE, the first trigger input is active
	gA[x]_DriveStatus.Trigger2				: If TRUE, the second trigger input is active
	gA[x]_DriveStatus.DriveEnable			: If TRUE, the enable input is active
	gA[x]_DriveStatus.ControllerReady		: If TRUE, the controller is ready to beturned on
	gA[x]_DriveStatus.ControllerStatus		: If TRUE, the controller is turned on (Same as MC_Power.Status)
	gA[x]_DriveStatus.AxisError				: If TRUE, at least one error has occurred (not acknowledged)
	gA[x]_DriveStatus.LagWarning			: If TRUE, the lag error has exceeded the limit value specified for a warning*)
		MC_BR_ReadDriveStatus_0.Enable := 1;
		MC_BR_ReadDriveStatus_0.Axis := gA[15].Ident;
		MC_BR_ReadDriveStatus_0.AdrDriveStatus := ADR (DriveStatus);
		MC_BR_ReadDriveStatus_0();
		gA[15].Ind_Simulation		:=	DriveStatus.Simulation;
		gA[15].Ind_NetworkInit		:=	DriveStatus.NetworkInit;
		gA[15].Input_Home			:=	DriveStatus.HomeSwitch;
		gA[15].Input_PosHW			:=	DriveStatus.PosHWSwitch;
		gA[15].Input_NegHW			:=	DriveStatus.NegHWSwitch;
		gA[15].Input_Trigger1		:=	DriveStatus.Trigger1;
		gA[15].Input_Trigger2		:=	DriveStatus.Trigger2;
		gA[15].Input_DriveEnable		:=	DriveStatus.DriveEnable;
		gA[15].Ind_ControllerReady	:=	DriveStatus.ControllerReady;
		gA[15].Ind_ControllerStatus	:=	DriveStatus.ControllerStatus;
		gA[15].Error					:=	DriveStatus.AxisError;
		gA[15].Ind_LagWarning		:=	DriveStatus.LagWarning;

	//*********************** READ AXIS ERROR *********************
		MC_ReadAxisError_0.Enable := gA[15].Ind_NetworkInit;
		MC_ReadAxisError_0.Axis := gA[15].Ident;
		MC_ReadAxisError_0.DataAddress := ADR(gA[15].ErrorText);
		MC_ReadAxisError_0.DataLength := SIZEOF(gA[15].ErrorText);
		MC_ReadAxisError_0.DataObjectName := 'Error_Eng';
		MC_ReadAxisError_0();
		IF(MC_ReadAxisError_0.Valid) THEN
			gA[15].ErrorID := MC_ReadAxisError_0.AxisErrorID;
			gA[15].ErrorCount := MC_ReadAxisError_0.AxisErrorCount;
		END_IF
	// Auto Acknowledge Errors
		IF (gA[15].Cmd_Reset AND (gA[15].ErrorCount<>0) AND NOT AutoAck) THEN
			AutoAck:=1;
		ELSE
			AutoAck:=0;
		END_IF
	//Axis Error Acknowledge
		IF (EDGEPOS(AutoAck) OR EDGEPOS(gA[15].ErrorAck)) THEN
			MC_ReadAxisError_0.Acknowledge := 1;
		ELSE;
			MC_ReadAxisError_0.Acknowledge :=0;
		END_IF

	//*********************** RESET AXIS ERROR *********************
		IF (gA[15].Cmd_Reset AND (gA[15].ErrorCount=0) AND gA[15].ErrorStop) THEN
			MC_Reset_0.Execute:=1;
		END_IF
		IF (MC_Reset_0.Done) THEN
			MC_Reset_0.Execute:=0;
			gA[15].Cmd_Reset:=0;
			ResetError := 0;
		END_IF
		IF (MC_Reset_0.Error) THEN
			MC_Reset_0.Execute:=0;
			gA[15].Cmd_Reset:=0;
			ResetError := 1;
		END_IF
		MC_Reset_0.Axis:=gA[15].Ident;
		MC_Reset_0();

	//*********************** READ AXIS STATUS ************************
		MC_ReadStatus_0.Enable := gA[15].Ind_NetworkInit;
		MC_ReadStatus_0.Axis := gA[15].Ident;
		MC_ReadStatus_0();
		IF(MC_ReadStatus_0.Valid = TRUE)THEN
			gA[15].Ind_Enabled 			:= NOT (MC_ReadStatus_0.Disabled);
			gA[15].Ind_StandStill		:= MC_ReadStatus_0.StandStill;
			gA[15].Ind_Stopping			:= MC_ReadStatus_0.Stopping;
			gA[15].Ind_DiscreteMotion	:= MC_ReadStatus_0.DiscreteMotion;
			gA[15].Ind_ContinuousMotion	:= MC_ReadStatus_0.ContinuousMotion;
			gA[15].Ind_SynchronizedMotion:= MC_ReadStatus_0.SynchronizedMotion;
			gA[15].ErrorStop				:= MC_ReadStatus_0.Errorstop;
		END_IF

	//******************* INIT POSITION MODULUS  ********************
    IF (g_rNumbPliers <> 0.0) THEN
      IF ( gA[15].Ind_StandStill     OR
           NOT(gA[15].Ind_Enabled) ) AND
         g_bChangeModDrumReq        THEN
        bChangeModReq := 1 ;
        uiInitModPos0_ErrorID := 0 ;
      END_IF
      MC_BR_InitModPos_0.Execute:= (InitModPosition OR bChangeModReq) ;
  		MC_BR_InitModPos_0.Axis:= gA[15].Ident;
  		MC_BR_InitModPos_0.Period:= REAL_TO_UDINT(gA[15].AxisPeriod * 4.0/g_rNumbPliers);
  		MC_BR_InitModPos_0.Factor:=1;
  		InitModPos_Done:=MC_BR_InitModPos_0.Done;
    END_IF
    IF MC_BR_InitModPos_0.Done THEN
      g_bChangeModDrumReq := 0 ;
      bChangeModReq       := 0 ;
    ELSIF MC_BR_InitModPos_0.Error THEN
      bChangeModReq := 0 ;
      uiInitModPos0_ErrorID := MC_BR_InitModPos_0.ErrorID ;
    END_IF
		MC_BR_InitModPos_0();

	//******************* INIT ENDLESS POSITION ********************
		MC_BR_InitEndlessPosition_0.Execute:= InitModPos_Done;
		MC_BR_InitEndlessPosition_0.Axis:= gA[15].Ident;
		MC_BR_InitEndlessPosition_0.DataAddress:= ADR(gEndPosData[15]);
		IF (MC_BR_InitEndlessPosition_0.Done) THEN
			InitModPosition:=0;
			InitEndlessPosition:=0;
			HomeRestore:=1;
		END_IF
		MC_BR_InitEndlessPosition_0();

	//*********************** HOME AXIS FIRST POWER UP *********************
		IF (HomeRestore AND NOT gA15_FirstHomed) THEN
			MC_Home_0.Execute:=1;
		END_IF
		MC_Home_0.Axis:=gA[15].Ident;
		MC_Home_0.Position:=0;
		MC_Home_0.HomingMode:=mcHOME_DIRECT;
		IF (MC_Home_0.Done) THEN
			MC_Home_0.Execute:=0;
			gA15_FirstHomed:=1;
		END_IF
		MC_Home_0();

	//*********************** HOME AXIS *********************
		IF (gA15_FirstHomed) THEN
			MC_Home_1.Execute:=HomeRestore;
		END_IF
		MC_Home_1.Axis:=gA[15].Ident;
		MC_Home_1.Position:=0;
		MC_Home_1.HomingMode:=mcHOME_RESTORE_POS;
		IF (MC_Home_1.Done) THEN
			gA[15].Ind_Homed:=1;
			HomeRestore:=0;
		END_IF
		MC_Home_1();

	//******************* READ ACTUAL POSITION ********************
		MC_ReadActualPosition_0.Enable:= gA[15].Ind_NetworkInit;
		MC_ReadActualPosition_0.Axis:= gA[15].Ident;
		MC_ReadActualPosition_0();
		IF(MC_ReadActualPosition_0.Valid = TRUE)THEN
			gA[15].PositionCount := MC_ReadActualPosition_0.Position;
			gA[15].PositionInch := gA[15].PositionCount/gA[15].UnitsPerInch;
			gA[15].PositionDeg := gA[15].PositionCount/gA[15].UnitsPerDeg;
		END_IF

  //******************** READ SET POINT POSITION *********************
    // Slave side  : ParID 428 SGEN_S_SET : CTRL Position controller: Input set position
    // Master side : ParID 412 S_SET_VAX1 : 412: VAX: Position

    // Slave side
    MC_BR_CyclicRead_0.Axis        := gA[15].Ident ;
    MC_BR_CyclicRead_0.Enable      := gA[15].Ind_NetworkInit;
    MC_BR_CyclicRead_0.ParID       := 428 ;
    MC_BR_CyclicRead_0.DataAddress := ADR(iiSP_SlPos_U);
    MC_BR_CyclicRead_0.DataType    := ncPAR_TYP_DINT ;
    // Master side
    MC_BR_CyclicRead_1.Axis        := gA[9].Ident ;
    MC_BR_CyclicRead_1.Enable      := gA[15].Ind_NetworkInit;
    MC_BR_CyclicRead_1.ParID       := 412 ;
    MC_BR_CyclicRead_1.DataAddress := ADR(iiSP_MaPos_U);
    MC_BR_CyclicRead_1.DataType    := ncPAR_TYP_DINT ;

    IF MC_BR_CyclicRead_0.Valid THEN
      rSP_SlPos_Deg := iiSP_SlPos_U/gA[15].UnitsPerDeg ;
      g_rTest_[1] := rSP_SlPos_Deg - TRUNC(rSP_SlPos_Deg/360.0)*360.0 ;
      g_rTest_[2] := g_rTest_[1] - gA[15].PositionDeg ;
    ELSIF MC_BR_CyclicRead_0.Error THEN
      MC_BR_CyclicRead_0.Enable := 0 ;
    END_IF
    IF MC_BR_CyclicRead_1.Valid THEN
      rSP_MaPos_Deg := iiSP_MaPos_U/gA[9].UnitsPerDeg ;
      g_rTest_[3] := rSP_MaPos_Deg - TRUNC(rSP_MaPos_Deg/360.0)*360.0 ;
      g_rTest_[4] := g_rTest_[3] - gA[9].PositionDeg ;
    ELSIF MC_BR_CyclicRead_1.Error THEN
      MC_BR_CyclicRead_1.Enable := 0 ;
    END_IF
    MC_BR_CyclicRead_0();
    MC_BR_CyclicRead_1();

  //******************** READ ACTUAL OFFSET *********************
  IF gA[15].rRSynDen > 0.0 THEN
    rTempActPhasDeg := rSP_SlPos_Deg - gA[15].rRSynNum / gA[15].rRSynDen * rSP_MaPos_Deg ;
    gA[15].rActPhasDeg := H_FC_Modulus (
                              IN_rMod := 360 * gA[15].rRSynNum / gA[15].rRSynDen ,
                              IN_rVar := rTempActPhasDeg
                                      ) ;
  END_IF

	//******************* READ ACTUAL VELOCITY ********************
		IF(MC_ReadActualVelocity_0.Error=TRUE) THEN
			MC_ReadActualVelocity_0.Enable:= 0;
		ELSE
			MC_ReadActualVelocity_0.Enable:= 1;
		END_IF
		MC_ReadActualVelocity_0.Axis:= gA[15].Ident;
		MC_ReadActualVelocity_0();
		IF(MC_ReadActualVelocity_0.Valid = TRUE)THEN
			//gA[15].ActualVelocity := MC_ReadActualVelocity_0.Velocity*60/gA[15].SP_MotorPPR;
      gA[15].ActualVelocity := MC_ReadActualVelocity_0.Velocity*60/gA[15].AxisPeriod ; // D.M. 03/08/2011 BrownPaper_14542  Need speed of the axis and not of the shaft of the motor
      IF ABS(gA[15].ActualVelocity>1) THEN // D.M. 03/08/2011 BrownPaper_14542 Add ABS because in case negative velocity Ind_InMotion = 0 instead of 1
				gA[15].Ind_InMotion:=1;
			ELSE
				gA[15].Ind_InMotion:=0;
			END_IF
		END_IF

	//******************* READ ACTUAL TORQUE ********************
		IF(MC_ReadActualTorque_0.Error=TRUE) THEN
			MC_ReadActualTorque_0.Enable:= 0;
		ELSE
			MC_ReadActualTorque_0.Enable:= 1;
		END_IF
		MC_ReadActualTorque_0.Axis:= gA[15].Ident;
		MC_ReadActualTorque_0();
		IF(MC_ReadActualTorque_0.Valid = TRUE)THEN
			gA[15].ActualTorque := MC_ReadActualTorque_0.Torque;
		END_IF

	//*********************** ENABLE AXIS *********************
		MC_Power_0.Axis:=gA[15].Ident;
		IF (MC_Power_0.Error=0) THEN
      MC_Power_0.Enable:=gA[15].Cmd_Enable OR bTest_[0];
		ELSE;
			MC_Power_0.Enable:=0;
		END_IF;
		MC_Power_0();

	//*********************** AXIS VELOCITY MOVE *********************
		MC_MoveVelocity_0.Axis         := gA[15].Ident;
		MC_MoveVelocity_0.Velocity     := g_stHMPerfCyc.rSP_Vel * gA[15].AxisPeriod/60;
		MC_MoveVelocity_0.Acceleration := g_stHMPerfCyc.rSP_Acc * gA[15].AxisPeriod/60/60;
		MC_MoveVelocity_0.Deceleration := g_stHMPerfCyc.rSP_Dec * gA[15].AxisPeriod/60/60;
		MC_MoveVelocity_0.Direction    := mcPOSITIVE_DIR;
	  MC_MoveVelocity_0.Execute      := g_stHMPerfCyc.Cmd_SlowRot;

    IF (MC_MoveVelocity_0.InVelocity)  OR
       (MC_MoveVelocity_0.Error)       OR
       g_stHMPerfCyc.Cmd_Stop          THEN
      g_stHMPerfCyc.Cmd_SlowRot := 0 OR bTest_[1] ;
    END_IF
		MC_MoveVelocity_0();

  //************************ AXIS HALT **********************
    MC_Halt_0.Axis := gA[15].Ident ;
    MC_Halt_0.Deceleration := g_stHMPerfCyc.rSP_Dec * gA[15].AxisPeriod/60/60;
    IF g_stHMPerfCyc.Cmd_Stop THEN
      MC_Halt_0.Execute := 1 ;
    END_IF
    IF (MC_Halt_0.Done)  OR
       (MC_Halt_0.Error) THEN
      MC_Halt_0.Execute := 0 ;
      g_stHMPerfCyc.Cmd_Stop := 0 ;
    END_IF
    MC_Halt_0();

  //************************ AXIS OVERRIDE **********************
    MC_SetOverride_0.Axis      := gA[15].Ident ;
    MC_SetOverride_0.Enable    := gA[15].Cmd_Override ;
    MC_SetOverride_0.VelFactor := gA[15].rSP_OverrideV ;
    MC_SetOverride_0.AccFactor := gA[15].rSP_OverrideA ;
    IF (MC_SetOverride_0.Enabled) OR
       (MC_SetOverride_0.Error)   THEN
      gA[15].Cmd_Override := 0 ;
    END_IF
    MC_SetOverride_0();

	//*********************** AXIS STOP *********************
		MC_Stop_0.Axis:=gA[15].Ident;
    //IF (gA[15].Ind_ContinuousMotion AND (NOT gA[15].Cmd_ContinuousMotion) AND gAlarmsOK) THEN
    IF FALSE THEN
			MC_Stop_0.Deceleration:=gA[15].SP_Decel;
			MC_Stop_0.Execute:=1;
		END_IF;
		IF (MC_Stop_0.Done OR MC_Stop_0.CommandAborted OR MC_Stop_0.Error) THEN
			MC_Stop_0.Execute:=0;
		END_IF;
		MC_Stop_0();

  //***********************  ESTOP *********************
    MC_Stop_1.Axis:=gA[15].Ident;
    IF EDGEPOS(g_bIndEStopStandstill) THEN
      MC_Stop_1.Deceleration:=gA[15].SP_EStopDecel;
      MC_Stop_1.Execute:=1;
    END_IF;
    IF (MC_Stop_1.Done OR MC_Stop_1.CommandAborted OR MC_Stop_1.Error) THEN
      MC_Stop_1.Execute:=0;
      gA[15].Cmd_EStopDisable := 1 ;
    END_IF;
    IF NOT(g_bIndEStopStandstill) THEN
      gA[15].Cmd_EStopDisable := 0 ;
    END_IF;
    MC_Stop_1();

		//*********************** AXIS PHASE CONTROL (Inches) *********************
    IF gA[15].Cmd_PhaseOffset OR
       g_bHMP_CmdPhasing      THEN
      rSP_PhaseOffset := gA[15].SP_PhaseOffset ;
      IF g_bHMP_CmdPhasing THEN
        g_bHMP_CmdPhasing    := 0 ;
        g_bHMP_PhasInProgres := 1 ;
        rSP_PhaseOffset := g_rHMP_SP_Phasing/360.0 * gRecipeActive.Repeat ;
      END_IF
      bCmd_PhaseOffset := 1 ;
    END_IF

		MC_BR_Phasing_0.Slave:=gA[15].Ident;
		IF gA[15].Ind_SynchronizedMotion AND NOT(gstCycA[7].CycManTimSet.bSCyc) AND st_TON_0.Q THEN
			MC_BR_Phasing_0.Enable:=1;
		ELSE;
			MC_BR_Phasing_0.Enable:=0;
		END_IF;
    IF bCmd_PhaseOffset AND NOT(gstCycA[7].CycManTimSet.bSCyc) THEN
			MC_BR_Phasing_0.InitData:=1;
      bCmd_PhaseOffset := 0 ;
      // Calculation new phase Drum/Master
      rTemp_[4] := rSP_PhaseOffset/gA[15].InchPerDeg ;
      rTemp_[5] := gRecipeActive.rHMPerf_PhasMasterDeg + rTemp_[4]*gA[15].rRSynNum/gA[15].rRSynDen ;
      gRecipeActive.rHMPerf_PhasMasterDeg := H_FC_Modulus (IN_rMod := 360, IN_rVar := rTemp_[5]) ;
      iTest_[2] := iTest_[2] + 1 ;
		ELSE
			MC_BR_Phasing_0.InitData:=0;
		END_IF
		MC_BR_Phasing_0.Shift               := rSP_PhaseOffset*gA[9].UnitsPerInch;
		MC_BR_Phasing_0.Velocity            := 6*gA[15].AxisPeriod/60;
		MC_BR_Phasing_0.Acceleration        := gA[15].SP_Decel;
		MC_BR_Phasing_0.ApplicationDistance := 0.8*gA[9].AxisPeriod * gA[15].rRSynNum/gA[15].rRSynDen ;
    MC_BR_Phasing_0.ApplicationMode     := mcTIME_BASED ; //mcMASTER_DISTANCE_BASED;
		MC_BR_Phasing_0.ShiftMode           := mcRELATIVE;
		MC_BR_Phasing_0();

    IF MC_BR_Phasing_0.ShiftAttained THEN
      g_bHMP_PhasInProgres   := 0 ;
      gA[15].Cmd_PhaseOffset := 0 ;
    END_IF

    //*********************** AXIS PHASE CONTROL (Inches) TIMING SETTING *********************
    IF gstCycA[7].CycManTimSet.bSCyc THEN
      IF gA[15].Cmd_ManuTimSetPlus THEN
        rAxisTimSet_SP_Vel := gr_rAxisTimSet_SP_Vel*gA[9].AxisPeriod/60 / (gA[15].rRSynNum/gA[15].rRSynDen) ;
      ELSE
        rAxisTimSet_SP_Vel := - gr_rAxisTimSet_SP_Vel*gA[9].AxisPeriod/60 / (gA[15].rRSynNum/gA[15].rRSynDen) ;
      END_IF
        rAxisTimSet_SP_Acc := gr_rAxisTimSet_SP_Acc*gA[9].AxisPeriod/60/60 ;
    END_IF

    MC_BR_Phasing_1.Slave                  := gA[15].Ident;
    MC_BR_Phasing_1.Enable                 := gstCycA[7].CycManTimSet.bCyc ;
    MC_BR_Phasing_1.InitData               := gstCycA[7].CycManTimSet.bSCyc ;
    MC_BR_Phasing_1.PerformVelocityControl := gstCycA[7].CycManTimSet.CmdMov ;
    MC_BR_Phasing_1.Velocity               := rAxisTimSet_SP_Vel ;
    MC_BR_Phasing_1.Acceleration           := rAxisTimSet_SP_Acc ;
    MC_BR_Phasing_1.ApplicationMode        := mcVELOCITY_CONTROL ;
    MC_BR_Phasing_1();
    st_TON_0(IN:=NOT(MC_BR_Phasing_1.Enable),PT:=T#100ms) ;

    IF NOT(gstCycA[7].CycManTimSet.CmdMov) AND
       MC_BR_Phasing_1.ShiftAttained       OR
       NOT(gstCycA[7].CycManTimSet.bCyc)   OR
       MC_BR_Phasing_1.Error               AND
       1                                   THEN
      gstCycA[7].CycManTimSet.CmdStop := 0 ;
    END_IF

	END_IF

END_PROGRAM
```

### Program Logical/BagMachine_Section/HotMicroPerf/Axis15/A15_Control (IEC) - Servo Control

#### A15_ControlCyclic.ld - Cyclic code
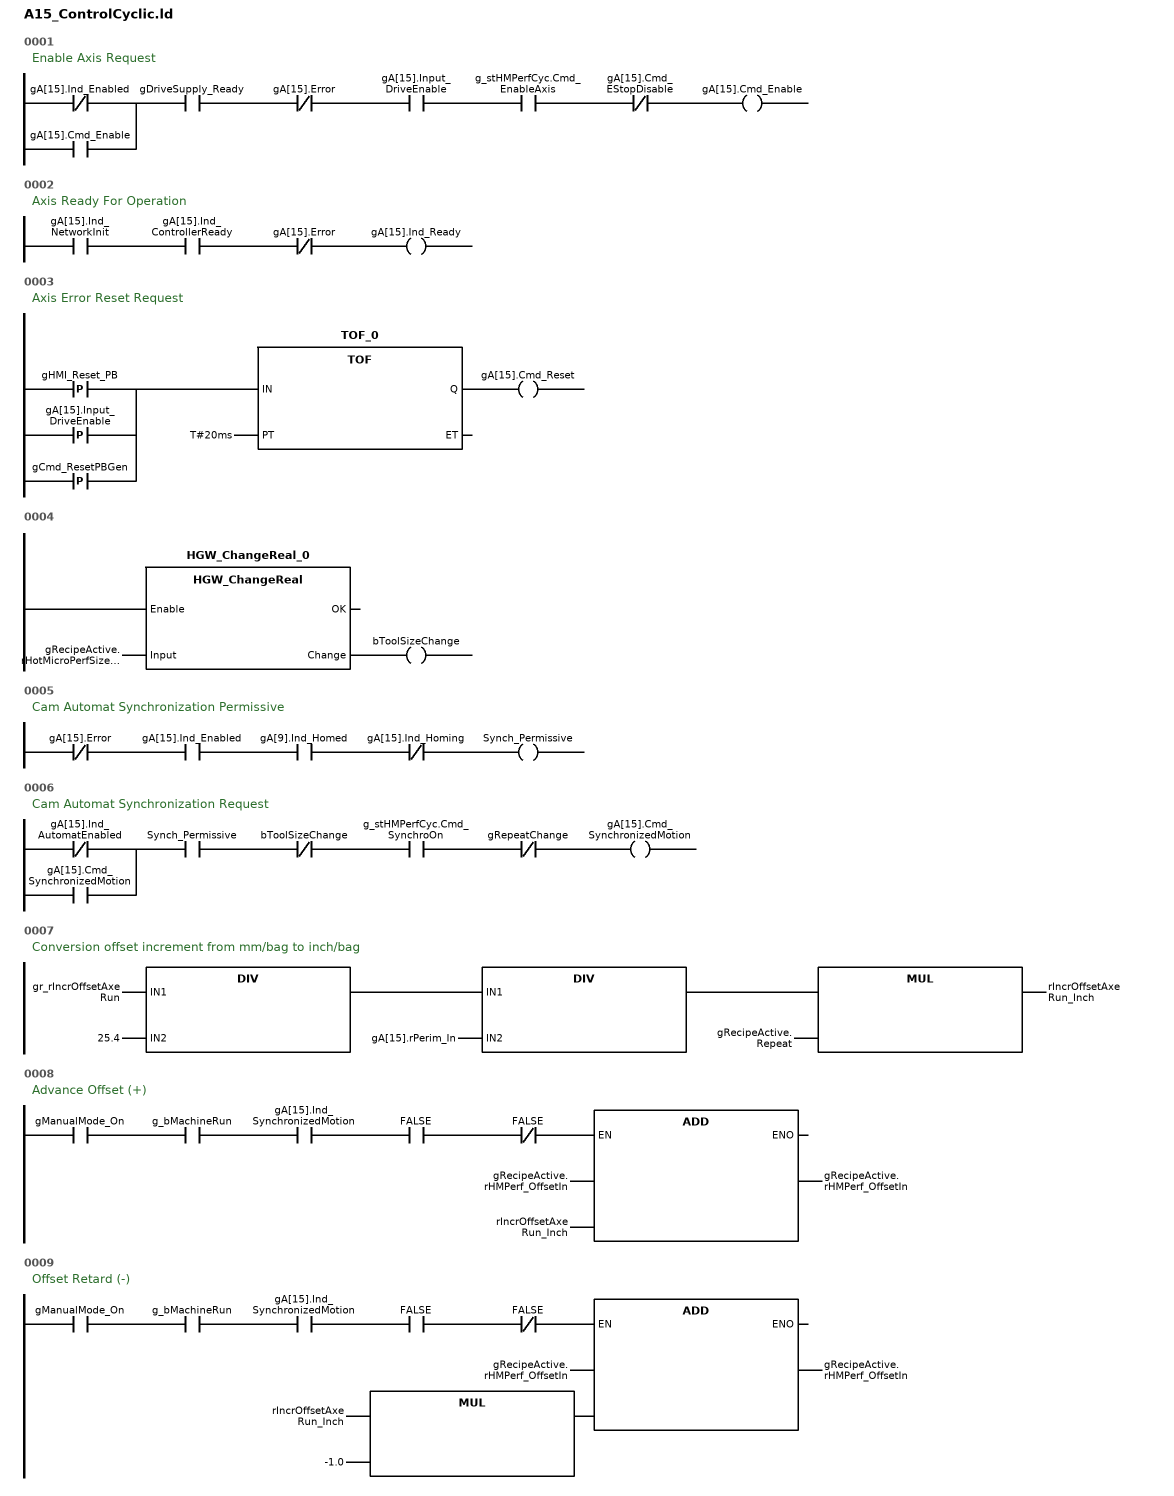
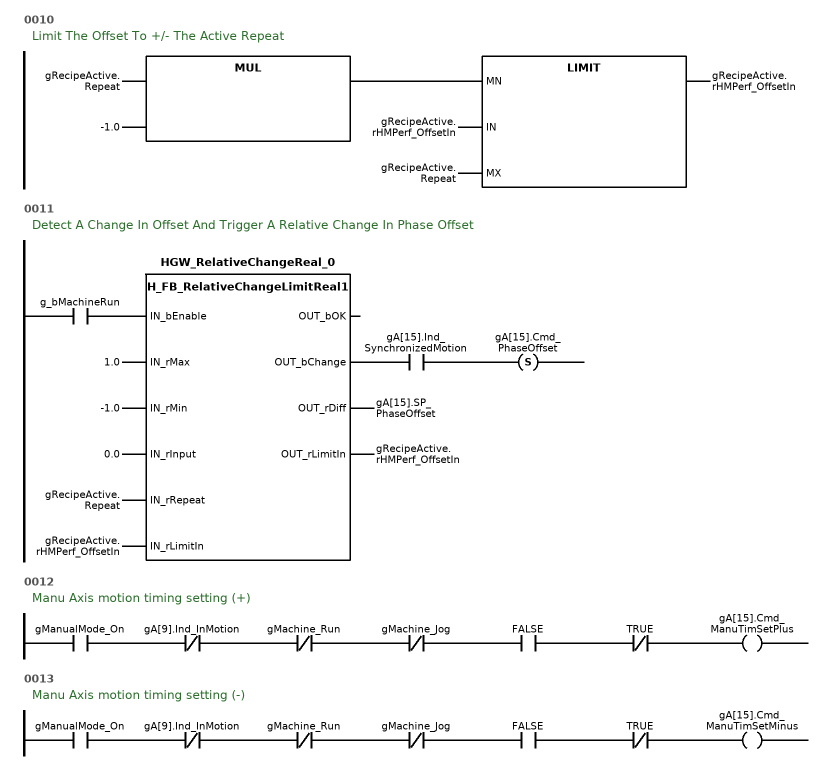
Ladder, written as Structured Text:
```iecst
(********************************************************************
 * COPYRIGHT -- Microsoft
 ********************************************************************
 * Program: A7_Control
 * File: A7_ControlCyclic.ld
 * Author: pkiel
 * Created: July 13, 2011
 ********************************************************************
 * Implementation of program A7_Control
 ********************************************************************)

PROGRAM _CYCLIC
VAR
    _e1 : R_TRIG;
    _e2 : R_TRIG;
    _e3 : R_TRIG;
END_VAR
(* Network 1: Enable Axis Request *)
gA[15].Cmd_Enable := (NOT gA[15].Ind_Enabled OR gA[15].Cmd_Enable) AND gDriveSupply_Ready AND NOT gA[15].Error AND gA[15].Input_DriveEnable AND g_stHMPerfCyc.Cmd_EnableAxis AND NOT gA[15].Cmd_EStopDisable;

(* Network 2: Axis Ready For Operation *)
gA[15].Ind_Ready := gA[15].Ind_NetworkInit AND gA[15].Ind_ControllerReady AND NOT gA[15].Error;

(* Network 3: Axis Error Reset Request *)
_e1(CLK := gHMI_Reset_PB);
_e2(CLK := gA[15].Input_DriveEnable);
_e3(CLK := gCmd_ResetPBGen);
TOF_0(IN := _e1.Q OR _e2.Q OR _e3.Q, PT := T#20ms);
gA[15].Cmd_Reset := TOF_0.Q;

(* Network 4 *)
HGW_ChangeReal_0(Enable := TRUE, Input := gRecipeActive.rHotMicroPerfSize_in);
bToolSizeChange := HGW_ChangeReal_0.Change;

(* Network 5: Cam Automat Synchronization Permissive *)
Synch_Permissive := NOT gA[15].Error AND gA[15].Ind_Enabled AND gA[9].Ind_Homed AND NOT gA[15].Ind_Homing;

(* Network 6: Cam Automat Synchronization Request *)
gA[15].Cmd_SynchronizedMotion := (NOT gA[15].Ind_AutomatEnabled OR gA[15].Cmd_SynchronizedMotion) AND Synch_Permissive AND NOT bToolSizeChange AND g_stHMPerfCyc.Cmd_SynchroOn AND NOT gRepeatChange;

(* Network 7: Conversion offset increment from mm/bag to inch/bag *)
rIncrOffsetAxeRun_Inch := ((gr_rIncrOffsetAxeRun / 25.4) / gA[15].rPerim_In) * gRecipeActive.Repeat;

(* Network 8: Advance Offset (+) *)
(* never executed: gRecipeActive.rHMPerf_OffsetIn := gRecipeActive.rHMPerf_OffsetIn + rIncrOffsetAxeRun_Inch; *)

(* Network 9: Offset Retard (-) *)
(* never executed: gRecipeActive.rHMPerf_OffsetIn := gRecipeActive.rHMPerf_OffsetIn + (rIncrOffsetAxeRun_Inch * -1.0); *)

(* Network 10: Limit The Offset To +/- The Active Repeat *)
gRecipeActive.rHMPerf_OffsetIn := LIMIT(MN := gRecipeActive.Repeat * -1.0, IN := gRecipeActive.rHMPerf_OffsetIn, MX := gRecipeActive.Repeat);

(* Network 11: Detect A Change In Offset And Trigger A Relative Change In Phase Offset *)
HGW_RelativeChangeReal_0(IN_bEnable := g_bMachineRun, IN_rMax := 1.0, IN_rMin := -1.0, IN_rInput := 0.0, IN_rRepeat := gRecipeActive.Repeat, IN_rLimitIn := gRecipeActive.rHMPerf_OffsetIn);
IF HGW_RelativeChangeReal_0.OUT_bChange AND gA[15].Ind_SynchronizedMotion THEN
    gA[15].Cmd_PhaseOffset := TRUE;
END_IF;
gA[15].SP_PhaseOffset := HGW_RelativeChangeReal_0.OUT_rDiff;
gRecipeActive.rHMPerf_OffsetIn := HGW_RelativeChangeReal_0.OUT_rLimitIn;

(* Network 12: Manu Axis motion timing setting (+) *)
gA[15].Cmd_ManuTimSetPlus := FALSE;

(* Network 13: Manu Axis motion timing setting (-) *)
gA[15].Cmd_ManuTimSetMinus := FALSE;
END_PROGRAM
```

### Program Logical/BagMachine_Section/HotMicroPerf/Axis15/A15_Automat (IEC) - Cam Automat

#### A15_Automat.var
```iecst
(********************************************************************
 * COPYRIGHT -- Microsoft
 ********************************************************************
 * Program: A15_Automat
 * File: A15_Automat.var
 * Author: dominique
 * Created: November 03, 2011
 ********************************************************************
 * Local variables of program A15_Automat
 ********************************************************************)
VAR
	AutData : MC_AUTDATA_TYP;
	AutomatStart : BOOL;
	ErrorID : UINT;
	MasterOffset : REAL;
  MasterParID : UINT;
  uiMasterParID1 : UINT;
	MC_BR_AutControl_0 : MC_BR_AutControl;
  MC_BR_InitMasterParIDTransfer_0 : MC_BR_InitMasterParIDTransfer;
  ParID_Ready : BOOL;
	PositionMOD : DINT;
	PositionOffset : DINT;
	SlaveStartOffset : REAL;
	Synch_Request : BOOL;
  uiSP_MasterParID : UINT;
  uiiSP_Master : UDINT;
  uiiSlaveFactor : UDINT;
  uiiMasterFactor : UDINT;
  usiMemoStat : USINT ;
  iiMasterFactor5 : DINT;
  iiSlaveFactor5  : DINT;
  bCmdSynchroOn : BOOL ;
  bCmdSynchroOff : BOOL ;
  rMaCompDist : REAL ;
  rSPMaPos    : REAL ;
  rOffsetDeg  : REAL ;
  rSlCompDist : REAL ;
  rTemp_      : ARRAY[0..9] OF REAL ;
  rRepeatMetric : REAL;
  rSlave_AxisPeriod : REAL ;
  rMaster_AxisPeriod : REAL ;
  bTest : BOOL ;
END_VAR
```

#### A15_AutomatCyclic.st
```iecst
(********************************************************************
 * COPYRIGHT -- Microsoft
 ********************************************************************
 * Program: A15_Automat
 * File: A15_AutomatCyclic.st
 * Author: dominique
 * Created: November 03, 2011
 ********************************************************************
 * Implementation of program A15_Automat
 ********************************************************************)

PROGRAM _CYCLIC

(**** STRAIGHT GEARED CAM AUTOMAT WITH ABSOLUTE PHASE SYNCHRONIZATION FOR DRUM ***)

  MC_BR_AutControl_0.Signal1 := (MC_BR_AutControl_0.ActualStateIndex=0) ;

  MC_BR_AutControl_0.Signal3 := g_stHMPerfCyc.Cmd_SynchroOff ;
  IF g_stHMPerfCyc.Cmd_SynchroOff            AND
     (MC_BR_AutControl_0.ActualStateIndex=4) THEN
    g_stHMPerfCyc.Cmd_SynchroOn  := 0 ;
    g_stHMPerfCyc.Cmd_SynchroOff := 0 ;
  END_IF

  // Synchro OK indicator
  gstCycA[15].CycManTimSet.bSynchroOkSlavA[15] := ( MC_BR_InitMasterParIDTransfer_0.MasterParID = gstCycA[15].CycManTimSet.uiMasterParID ) AND
                                                  ( MC_BR_AutControl_0.ActualStateIndex = 4 )                                              AND
                                                  gA[15].Ind_SynchronizedMotion AND ParID_Ready ;
  gstCycA[15].CycManTimSet.bSynchroOkSlavA[15] := gstCycA[15].CycManTimSet.bSynchroOkSlavA[15] ;

	Synch_Request := gA[15].Cmd_SynchronizedMotion;
	IF (Synch_Request AND NOT ParID_Ready) THEN
	  MC_BR_InitMasterParIDTransfer_0.Master:= gA[9].Ident ;
    MC_BR_InitMasterParIDTransfer_0.Slave:= gA[15].Ident ;
    MC_BR_InitMasterParIDTransfer_0.MasterParID:= 412 ; // ParID 412 = 412: VAX: Position (in case virtual axis)
    MC_BR_InitMasterParIDTransfer_0.SlaveChannel:=0;
    MC_BR_InitMasterParIDTransfer_0.Execute:=TRUE;
    IF (MC_BR_InitMasterParIDTransfer_0.Done) THEN
      MasterParID:=MC_BR_InitMasterParIDTransfer_0.ReceiveParID;
      MC_BR_InitMasterParIDTransfer_0.Execute:=FALSE;
      ParID_Ready:=1;
    ELSIF (MC_BR_InitMasterParIDTransfer_0.Error) THEN
    (*Store ErrorID in a variable,
      ErrorID is reset on falling edge of 'Execute'*)
      ErrorID:=MC_BR_InitMasterParIDTransfer_0.ErrorID;
      ParID_Ready:=0;
      MC_BR_InitMasterParIDTransfer_0.Execute:=FALSE;
    END_IF
	END_IF
  MC_BR_InitMasterParIDTransfer_0();

(**** Initialize Automat Parameters Upon Automat Start Request ****)
	IF (EDGEPOS(ParID_Ready))THEN

		(**** Calculate Slave Start Offset ****)
      MasterOffset := gRecipeActive.rHMPerf_OffsetIn ;
			PositionOffset:= REAL_TO_DINT((gA[9].PositionInch-(gA[15].PositionInch-MasterOffset))*1000);
			PositionMOD:= REAL_TO_DINT(gRecipeActive.Repeat*1000);
			SlaveStartOffset:= (DINT_TO_REAL(PositionOffset MOD PositionMOD))/1000;
			IF (SlaveStartOffset >= (0.5*gRecipeActive.Repeat)) THEN
				SlaveStartOffset := SlaveStartOffset - gRecipeActive.Repeat;
			END_IF
			IF (SlaveStartOffset < (-0.5*gRecipeActive.Repeat)) THEN
				SlaveStartOffset := SlaveStartOffset + gRecipeActive.Repeat;
      END_IF

    // Master Slave periode
    IF gRecipeActive.bHMPerf_Mode THEN
      // Case Interrupt
      rMaster_AxisPeriod := gA[9].AxisPeriod * gRecipeActive.iHMPerf_Up ;
      rSlave_AxisPeriod  := gA[15].AxisPeriod ;
    ELSE
      // Case Continu
      rMaster_AxisPeriod := gA[9].AxisPeriod * gA[15].rRSynDen ;
      rSlave_AxisPeriod  := gA[15].AxisPeriod * gA[15].rRSynNum ;
    END_IF

		(*general automat parameter*)
			(*AutData.Master			  	:= gA1.Ident;*)
			AutData.MasterParID	  		:= MasterParID;
			AutData.StartPosition  		:= 0;
			AutData.StartInterval	  	:= gA[9].AxisPeriod;
			AutData.MaxMasterVelocity	:= gr_rMachMaxSpeed_BPM ;

		(*Automat STATE 0 Basis State*)
			AutData.State[0].Event[0].Type		  := ncSIGNAL1;
			AutData.State[0].Event[0].Attribute	:= ncAT_ONCE;
      AutData.State[0].Event[0].NextState := 1;

      rTemp_[0] := gA[15].PositionDeg ;
      rTemp_[1] := gA[9].PositionDeg ;

    // Master/Slave synchro calculation
      rOffsetDeg := gRecipeActive.rHMPerf_OffsetIn/gRecipeActive.Repeat * 360.0 ;
      // Pos Master in Slave range
      rTemp_[2] := gA[15].rRSynNum/gA[15].rRSynDen * gA[9].PositionDeg ;
      // Slave distance to be synchronized
      rTemp_[3] := rTemp_[2] - gA[15].PositionDeg + rOffsetDeg ;
      rSlCompDist := rTemp_[3] ;
      IF rSlCompDist > 360 THEN
        rSlCompDist := rSlCompDist - 360.0 ;
      END_IF ;
      IF rSlCompDist < 0 THEN
        rSlCompDist := rSlCompDist + 360.0 ;
      END_IF ;

		//Automat STATE 1 Master/Slave Absolute Phase Correction
      AutData.State[1].MasterParID     := MasterParID ;
			AutData.State[1].CamProfileIndex := 16#FFFF;
			AutData.State[1].MasterFactor		 := REAL_TO_UDINT(rMaster_AxisPeriod*5);
      AutData.State[1].SlaveFactor     := REAL_TO_UDINT((rSlave_AxisPeriod*5)+(rSlCompDist*gA[15].UnitsPerDeg));
			AutData.State[1].CompMode			   := ncOFF;

      AutData.State[1].Event[0].Type      := ncST_END;
      AutData.State[1].Event[0].Attribute := ncST_END;
      AutData.State[1].Event[0].NextState := 3;

      AutData.State[1].Event[1].Type      := ncSIGNAL3;
      AutData.State[1].Event[1].Attribute := ncAT_ONCE;
      AutData.State[1].Event[1].NextState := 0;

    //Automat STATE 2 Master/Slave Transition
      (*AutData.State[2].CamProfileIndex    := 16#FFFF;
      AutData.State[2].MasterFactor       := REAL_TO_UDINT(rMaster_AxisPeriod);
      AutData.State[2].SlaveFactor        := REAL_TO_UDINT(rSlave_AxisPeriod);
      AutData.State[2].CompMode           := ncSL_ABS;
      AutData.State[2].MasterCompDistance := gA[9].AxisPeriod * 4 ;
      AutData.State[2].SlaveCompDistance  := gA[11].AxisPeriod ;
      AutData.State[2].ExtendedCompLimits := ncOFF;

      AutData.State[2].Event[0].Type      := ncST_END;
      AutData.State[2].Event[0].Attribute  := ncST_END;
      AutData.State[2].Event[0].NextState  := 3;*)

    //Automat STATE 3 Master/Slave Run
      AutData.State[3].MasterParID     := MasterParID ;
      AutData.State[3].CamProfileIndex := 16#FFFF;
      AutData.State[3].MasterFactor     := REAL_TO_UDINT(rMaster_AxisPeriod);
      AutData.State[3].SlaveFactor     := REAL_TO_UDINT(rSlave_AxisPeriod);
      AutData.State[3].CompMode         := ncOFF;

      AutData.State[3].Event[0].Type      := ncST_END;
      AutData.State[3].Event[0].Attribute  := ncST_END;
      AutData.State[3].Event[0].NextState  := 3;

      AutData.State[3].Event[1].Type      := ncST_END+ncNEGATIVE;
      AutData.State[3].Event[1].Attribute := ncST_END;
      AutData.State[3].Event[1].NextState := 3;

      AutData.State[3].Event[2].Type      := ncSIGNAL3;
      AutData.State[3].Event[2].Attribute := ncAT_ONCE;
      AutData.State[3].Event[2].NextState := 4;

    //Automat STATE 4 Stop
      AutData.State[4].MasterParID     := MasterParID ;
      AutData.State[4].CamProfileIndex := 16#FFFF;
      AutData.State[4].MasterFactor    := REAL_TO_UDINT(rMaster_AxisPeriod);
      AutData.State[4].SlaveFactor     := REAL_TO_UDINT(0.0);
      AutData.State[4].CompMode        := ncOFF;

      AutData.State[4].Event[0].Type       := ncAT_ONCE;
      AutData.State[4].Event[0].Attribute  := ncAT_ONCE;
      AutData.State[4].Event[0].NextState  := 0;

			MC_BR_AutControl_0.Enable 		 := 1;
			MC_BR_AutControl_0.AdrAutData  := ADR(AutData);
			MC_BR_AutControl_0.InitAutData := 1;
	END_IF
			(* wait for initialization done or restart *)
			IF ((MC_BR_AutControl_0.AutDataInitialized=1) AND (Synch_Request)) THEN
				MC_BR_AutControl_0.InitAutData := 0;
				MC_BR_AutControl_0.Enable :=1;
				AutomatStart := 1;;
			END_IF
			(* check if error occured *)
			IF (MC_BR_AutControl_0.ErrorID <> 0) THEN
				MC_BR_AutControl_0.Enable := 0;
			END_IF

	(******************** ENABLE CAM-AUTOMAT **********************)

	IF (AutomatStart) THEN
			MC_BR_AutControl_0.Start := 1;
			AutomatStart := 0;
	END_IF

	IF (NOT Synch_Request) THEN
			MC_BR_AutControl_0.Stop := 1;
			MC_BR_AutControl_0.Start := 0;
      ParID_Ready := 0;
			IF (MC_BR_AutControl_0.Running=0) THEN
				MC_BR_AutControl_0.Enable := 0;
				MC_BR_AutControl_0.Stop := 0;
			END_IF
	END_IF

	gA[15].Ind_AutomatEnabled:=MC_BR_AutControl_0.Enable;
	gA[15].Ind_CurrentAutomatState:=MC_BR_AutControl_0.ActualStateIndex;
  gA[15].Ind_bSynchroOK := (MC_BR_AutControl_0.ActualStateIndex = 3) AND gA[15].Ind_SynchronizedMotion ; ;

	(********************** MC_AUTCONTROL *************************)
	MC_BR_AutControl_0.Slave:= gA[15].Ident;
	MC_BR_AutControl_0();

END_PROGRAM
```

- Program Logical/BagMachine_Section/HotMicroPerf/Axis15/A15_Ref (IEC) - Reference Routine (no source held here)

### Program Logical/BagMachine_Section/HotMicroPerf/Axis15/A15_Cycle (IEC) - A new program

#### A15_Cycle.var - Local variables
```iecst
(********************************************************************
 * COPYRIGHT -- .
 ********************************************************************
 * Program: A15_Cycle
 * File: A15_Cycle.var
 * Author: dominique
 * Created: November 03, 2011
 ********************************************************************
 * Local variables of program A15_Cycle
 ********************************************************************)

VAR
  iTest_          : ARRAY [0..9] OF INT ;
  rTempActPhasDeg : ARRAY[0..9] OF REAL ;
  rTempActOffsetInch : ARRAY[0..9] OF REAL ;
  rTemp_          : ARRAY[0..9] OF REAL ;
  stTON_01        : TON ;

END_VAR

VAR CONSTANT

END_VAR
```

### Program Logical/BagMachine_Section/HotMicroPerf/Axis15/A15_MotionCycle (IEC) - Hot Micro Perf motion cycle

#### A15_MotionCycleCyclic.st
```iecst
(********************************************************************
 * COPYRIGHT -- .
 ********************************************************************
 * Program: A15_MotionCycle
 * File: A15_MotionCycleCyclic.st
 * Author: dominique
 * Created: November 06, 2011
 ********************************************************************
 * Implementation of program A15_MotionCycle
 ********************************************************************)

PROGRAM _CYCLIC
    // --------------------------------------------------------------------------------------------------------------------
    // Simul
    IF g_bSim THEN
      stTON_0(IN:=bQ_SOL_HMP_ProtecDown,PT:=T#3s) ;
      gI_HMP_ProtecDownPE := stTON_0.Q ;

      stTON_1(IN:=NOT(bQ_SOL_HMP_BrushForward),PT:=T#3s) ;
      gI_HMP_BrushReturnPE := stTON_1.Q ;
    END_IF ;

    //---------------------------------------------------------------------------------------------------------------------
    // Output assignment and manual mode
    IF NOT(g_stHMPerfCyc.bSelProd) THEN
      // Manu operation
      gQ_SOL_HMP_ProtecDown := gI_SS_HMP_ManuProtecDown   OR
                               gI_HMP_ManuBrushForward_PB OR
                               NOT(gI_HMP_BrushReturnPE)  ;

      gQ_SOL_HMP_BrushForward := gI_HMP_ManuBrushForward_PB AND
                                 gI_HMP_ProtecDownPE        ;
    ELSE
      // Automatic operation
      gQ_SOL_HMP_BrushForward := bQ_SOL_HMP_BrushForward AND
                                 gI_HMP_ProtecDownPE     ;
      gQ_SOL_HMP_ProtecDown := bQ_SOL_HMP_ProtecDown     OR
                               NOT(gI_HMP_BrushReturnPE) ;
    END_IF ;

    // Light indicator
    gQ_HMP_LightOn := g_stHMPerfCyc.bSelProd ;

    // Heater activation
    gQ_HMP_Heater := gI_SS_HMP_Heating             AND
                     g_stHMPerfCyc.bSelProd        AND
                     NOT(g_bIndEStop)              AND
                     g_bMainPower_On               AND
                     ( g_stHMPerfCyc.bSlowRot_OK   OR
                       g_stHMPerfCyc.bSynchro_OK ) ;

    //---------------------------------------------------------------------------------------------------------------------
    // Actual Line Speed, in m/min
    rLS_Act_mmin := gActualMachineSpeed_FPM/3.2808 + g_rTest_[0] ;

    //---------------------------------------------------------------------------------------------------------------------
    // Axis motion management cycle
    //---------------------------------------------------------------------------------------------------------------------
    // Start cycle
    IF g_stHMPerfCyc.bSelProd THEN
      g_stHMPerfCyc.bSCyc := 1 ;
    END_IF ;

    //----------------------------------------------------------------------
    // Cycle at rest
    IF NOT(g_stHMPerfCyc.bSCyc) AND
       1                        THEN
      IF NOT( g_stHMPerfCyc.bFCyc ) THEN
        // Init after cycle unpropaly ended
        g_stHMPerfCyc.bFCyc    := 1 ;
        g_stHMPerfCyc.bCyc     := 0 ;
        g_stHMPerfCyc.bCycFail := 1 ;

        g_stHMPerfCyc.Cmd_SlowRot    := 0 ;
        g_stHMPerfCyc.Cmd_Stop       := 0 ;
        g_stHMPerfCyc.Cmd_EnableAxis := 0 ;
        g_stHMPerfCyc.bSynchro_OK    := 0 ;
        g_stHMPerfCyc.bSlowRot_OK    := 0 ;
        gA[15].Cmd_CalcCameProf      := 0 ;
        g_bHMP_CmdPhasing            := 0 ;
        g_bHMP_PhasInProgres         := 0 ;
        bGearInError                 := 0 ;
        bQ_SOL_HMP_BrushForward      := 0 ;
        bQ_SOL_HMP_ProtecDown        := 0 ;
        g_stHMPerfCyc.bStopReq       := 0 ;
        g_stHMPerfCyc.bSelProd       := 0 ;
      END_IF
      g_stHMPerfCyc.iStep := 0 ;
      RETURN ;
    ELSE
    //----------------------------------------------------------------------
    // Cycle running

      // Permanent conditions

      // Reset fault
      IF gAlarmReset                     AND
         (g_stHMPerfCyc.iStep=C_iSTEP_2) THEN
        bGearInError := 0 ;
      END_IF

      // Fault conditions detection
      g_stHMPerfCyc.bFaultCond := NOT(gA[15].Ind_Ready)           OR
                                  gA[15].Cmd_EStopDisable         OR
                                  NOT(gA[15].Cmd_Enable)          AND
                                  g_stHMPerfCyc.Cmd_EnableAxis    OR
                                  bGearInError                    AND
                                  (g_stHMPerfCyc.iStep=C_iSTEP_0) ;

      // Stop conditions detection
      g_stHMPerfCyc.bStopCond := NOT(g_bMainPower_On)   OR
                                 bGearInError           OR
                                 g_stHMPerfCyc.bStopReq ;

      // Fault reaction
      IF g_stHMPerfCyc.bFaultCond AND
         g_stHMPerfCyc.bCyc       THEN
        g_stHMPerfCyc.iStep := C_iSTEP_2 ;

        g_stHMPerfCyc.Cmd_SlowRot    := 0 ;
        g_stHMPerfCyc.Cmd_Stop       := 0 ;
        g_stHMPerfCyc.Cmd_EnableAxis := 0 ;
        gA[15].Cmd_CalcCameProf      := 0 ;
        g_bHMP_CmdPhasing            := 0 ;
        g_bHMP_PhasInProgres         := 0 ;
        g_stHMPerfCyc.bSynchro_OK    := 0 ;
        g_stHMPerfCyc.bSlowRot_OK    := 0 ;
        bQ_SOL_HMP_BrushForward      := 0 ;
        bQ_SOL_HMP_ProtecDown        := 0 ;
      END_IF

      // Stop reaction
      IF g_stHMPerfCyc.bStopCond  AND
         g_stHMPerfCyc.bCyc       AND
         (g_stHMPerfCyc.iStep>4)  AND
         (g_stHMPerfCyc.iStep<15) THEN
        g_stHMPerfCyc.iStep := C_iSTEP_4 ;
        // Action Step 4
        // Waiting State
      END_IF

      // Permanent actions

      // Condition for Slow Rotation Detection
      g_stHMPerfCyc.bSlowRotCond := ( (rLS_Act_mmin<gr_rHMPerfSLActTool_mmin) OR
                                      gMachine_Jog )                          AND
                                    NOT(g_stHMPerfCyc.bSlowRot_OK)            ;

      // Synchro Axis
      MC_GearIn_0.Master           := gA[9].Ident ;  // Master Axis*)
      MC_GearIn_0.Slave            := gA[15].Ident ; // Slave Axis*)
      MC_GearIn_0.RatioNumerator   := 1 ;
      MC_GearIn_0.RatioDenominator := gRecipeActive.iHMPerf_Up ;
      MC_GearIn_0.Acceleration     := 1.5*gA[9].SP_Accel ;
      MC_GearIn_0.Deceleration     := 4*gA[9].SP_Decel ;
      IF MC_GearIn_0.InGear OR
         MC_GearIn_0.Error  THEN
        uiMC_GearIn_ErrorID := MC_GearIn_0.ErrorID ;
        bGearInError := MC_GearIn_0.Error ;
        MC_GearIn_0.Execute := 0 ;
      END_IF
      MC_GearIn_0() ;

    END_IF
    //----------------------------------------------------------------------
    // Cycle steps

        CASE g_stHMPerfCyc.iStep OF

        C_iSTEP_0 :
         //----------------------------------------------
         // Step 1 : Initialisation
         //----------------------------------------------
          IF TRUE THEN
            g_stHMPerfCyc.iStep := C_iSTEP_1 ;

            // Action Step 1
            g_stHMPerfCyc.bFCyc    := 0 ;
            g_stHMPerfCyc.bCyc     := 1 ;
            g_stHMPerfCyc.bCycFail := 0 ;

            g_stHMPerfCyc.bSynchro_OK := 0 ;
            g_stHMPerfCyc.bSlowRot_OK := 0 ;
          END_IF

        C_iSTEP_1 :
         //----------------------------------------------
         // Step 2  : Fault management
         // Step 3  : Enable Axis
         // Step 0  : First Step
         //----------------------------------------------
         // Conditions Step 2
          IF g_stHMPerfCyc.bFaultCond         AND
             ( g_stHMPerfCyc.bTestOn          OR
               NOT(g_stHMPerfCyc.bModTest) ) THEN
            g_stHMPerfCyc.iStep := C_iSTEP_4 ;

            // Action Step 2
            g_stHMPerfCyc.bTestOn := 0 ;

            // Fault management
            RETURN ;
          END_IF

         // Conditions Step 3
          IF gA[15].Ind_Ready                AND
             NOT(gA[15].Ind_Enabled)         AND
             NOT(g_stHMPerfCyc.bStopCond)    AND
             NOT(g_stHMPerfCyc.bFaultCond)   AND
             ( g_stHMPerfCyc.bTestOn         OR
               NOT(g_stHMPerfCyc.bModTest) ) THEN
            g_stHMPerfCyc.iStep := C_iSTEP_3 ;

            // Action Step 3
            g_stHMPerfCyc.bTestOn := 0 ;

            g_stHMPerfCyc.Cmd_EnableAxis := 1 ;
            RETURN ;
          END_IF

         // Conditions Step 0
          IF g_stHMPerfCyc.bStopReq           AND
             ( g_stHMPerfCyc.bTestOn          OR
               NOT(g_stHMPerfCyc.bModTest) ) THEN
            g_stHMPerfCyc.iStep := C_iSTEP_0 ;

            // Action Step 0
            g_stHMPerfCyc.bTestOn := 0 ;

            g_stHMPerfCyc.bSCyc := 0 ;
            g_stHMPerfCyc.bFCyc := 1 ;
            g_stHMPerfCyc.bCyc  := 0 ;

            g_stHMPerfCyc.bStopReq := 0 ;
            g_stHMPerfCyc.bSelProd := 0 ;
          END_IF

        C_iSTEP_2 :
         //----------------------------------------------
         // Step 4  : Waiting State
         // Step 3  : Enable Axis and Came calculation and Download
         // Step 0  : First Step
         //----------------------------------------------
         // Conditions Step 4
          IF gA[15].Ind_Enabled               AND
             NOT(g_stHMPerfCyc.bStopCond)     AND
             ( g_stHMPerfCyc.bTestOn          OR
               NOT(g_stHMPerfCyc.bModTest) ) THEN
            g_stHMPerfCyc.iStep := C_iSTEP_4 ;

            // Action Step 4
            g_stHMPerfCyc.bTestOn := 0 ;

            // Waiting State
            RETURN ;
          END_IF

         // Conditions Step 3
          IF gA[15].Ind_Ready                AND
             NOT(gA[15].Ind_Enabled)         AND
             NOT(g_stHMPerfCyc.bStopCond)    AND
             NOT(g_stHMPerfCyc.bFaultCond)   AND
             ( g_stHMPerfCyc.bTestOn         OR
               NOT(g_stHMPerfCyc.bModTest) ) THEN
            g_stHMPerfCyc.iStep := C_iSTEP_3 ;

            // Action Step 3
            g_stHMPerfCyc.bTestOn := 0 ;

            g_stHMPerfCyc.Cmd_EnableAxis := 1 ;
            RETURN ;
          END_IF

         // Conditions Step 0
          IF g_stHMPerfCyc.bStopCond          AND
             ( g_stHMPerfCyc.bTestOn          OR
               NOT(g_stHMPerfCyc.bModTest) ) THEN
            g_stHMPerfCyc.iStep := C_iSTEP_0 ;

            // Action Step 0
            g_stHMPerfCyc.bTestOn := 0 ;

            g_stHMPerfCyc.bSCyc := 0 ;
            g_stHMPerfCyc.bFCyc := 1 ;
            g_stHMPerfCyc.bCyc  := 0 ;

            g_stHMPerfCyc.bStopReq := 0 ;
            g_stHMPerfCyc.bSelProd := 0 ;
          END_IF

        C_iSTEP_3 :
         //----------------------------------------------
         // Step 4 : Waiting State
         //----------------------------------------------
          IF gA[15].Ind_Enabled THEN
            g_stHMPerfCyc.iStep := C_iSTEP_4 ;

            // Action Step 4
            // Waiting State
          END_IF

        C_iSTEP_4 :
         //----------------------------------------------
         // Step 15 : Stop request
         // Step 5  : Slow rotation    Return Brush
         // Step 10 : Synchro Axe
         //----------------------------------------------
         // Condititons Step 15
          IF g_stHMPerfCyc.bStopCond          AND
             ( g_stHMPerfCyc.bTestOn          OR
               NOT(g_stHMPerfCyc.bModTest) ) THEN
            g_stHMPerfCyc.iStep := C_iSTEP_15 ;

            // Action Step 15
            g_stHMPerfCyc.bTestOn := 0 ;

            RETURN ;
          END_IF

         // Condititons Step 5
          IF g_stHMPerfCyc.bSlowRotCond       AND
             ( g_stHMPerfCyc.bTestOn          OR
               NOT(g_stHMPerfCyc.bModTest) ) THEN
            g_stHMPerfCyc.iStep := C_iSTEP_5 ;

            // Action Step 5
            g_stHMPerfCyc.bTestOn := 0 ;

            // Return Brush
            bQ_SOL_HMP_BrushForward := 0 ;
            RETURN ;
          END_IF

         // Condititons Step 10
          IF NOT(g_stHMPerfCyc.bSynchro_OK)          AND
             (rLS_Act_mmin>gr_rHMPerfSLActTool_mmin) AND
             g_bMachineRun                           AND
             NOT(gA[15].Cmd_PhaseOffset)             AND
             ( g_stHMPerfCyc.bTestOn                 OR
               NOT(g_stHMPerfCyc.bModTest) )         THEN
            g_stHMPerfCyc.iStep := C_iSTEP_10 ;

            // Action Step 10
            g_stHMPerfCyc.bTestOn := 0 ;

            // Synchro Axe
            MC_GearIn_0.Execute       := 1 ;
            g_stHMPerfCyc.bSlowRot_OK := 0 ;
          END_IF

        C_iSTEP_5 :
         //----------------------------------------------
         // Step 6 : Move up protector
         //          Activate Slow Rotation
         //----------------------------------------------
          IF gI_HMP_BrushReturnPE             AND
             ( g_stHMPerfCyc.bTestOn          OR
               NOT(g_stHMPerfCyc.bModTest) ) THEN
            g_stHMPerfCyc.iStep := C_iSTEP_6 ;

            // Action Step 6
            g_stHMPerfCyc.bTestOn := 0 ;

            // Move down protector
            bQ_SOL_HMP_ProtecDown := 0 ;

            // Activate Slow Rotation
            g_stHMPerfCyc.bSlowRot_OK := 1 ;
            g_stHMPerfCyc.Cmd_SlowRot := 1 ;

            g_stHMPerfCyc.rSP_Vel := gr_rHMPerfSlowRot_rpm ;
            g_stHMPerfCyc.rSP_Acc := gr_rHMPerfAcc_rpm2 ;
            g_stHMPerfCyc.rSP_Dec := gr_rHMPerfDec_rpm2 ;
          END_IF

        C_iSTEP_6 :
         //----------------------------------------------
         // Step 7 : Synchro Off
         //----------------------------------------------
          IF NOT(gI_HMP_ProtecDownPE)           AND
             NOT(g_stHMPerfCyc.Cmd_SlowRot)     AND
             NOT(gA[15].Ind_SynchronizedMotion) AND
             ( g_stHMPerfCyc.bTestOn            OR
               NOT(g_stHMPerfCyc.bModTest) )   THEN
            g_stHMPerfCyc.iStep := C_iSTEP_7 ;

            // Action Step 7
            g_stHMPerfCyc.bTestOn := 0 ;

            g_stHMPerfCyc.bSynchro_OK := 0 ;
          END_IF

        C_iSTEP_7 :
         //----------------------------------------------
         // Step 4 : Waiting State
         //----------------------------------------------
          IF TRUE                              AND
             ( g_stHMPerfCyc.bTestOn           OR
               NOT(g_stHMPerfCyc.bModTest) )   THEN
            g_stHMPerfCyc.iStep := C_iSTEP_4 ;

            // Action Step 4
            g_stHMPerfCyc.bTestOn := 0 ;

            // Waiting State
          END_IF

        C_iSTEP_10 :
         //----------------------------------------------
         // Step 11 : Phasing
         //----------------------------------------------
          IF NOT(MC_GearIn_0.Execute)        AND
             ( g_stHMPerfCyc.bTestOn         OR
               NOT(g_stHMPerfCyc.bModTest) ) THEN
            g_stHMPerfCyc.iStep := C_iSTEP_11 ;

            // Action Step 11
            g_stHMPerfCyc.bTestOn := 0 ;

            // Synchro Phasing
            g_bHMP_CmdPhasing := 1 ;
            // Calculation Offset, in Deg
            rCalc[0] := (gRecipeActive.rHMPerf_OffsetIn + gRecipeActive.Perf_Offset) / gRecipeActive.Repeat * 360.0 ;
            // Calculation Actual Slave Phase on Master side, in Deg (PosSalve = R x PosMaster + Phase = R x ( PosMaster + Offset ) => Phase = R x Offset  with R = rRSynNum/rRSynDen
            rCalc[1] := gA[15].rActPhasDeg / (gA[15].rRSynNum/gA[15].rRSynDen) ;
            // Difference between Set Point Offset and Actual Offset
            rCalc[2] := rCalc[0] - rCalc[1] ;
            // Phase Shift Set Point to match with Set Point Offset
            g_rHMP_SP_Phasing := H_FC_Modulus (IN_rMod := 360.0, IN_rVar := rCalc[2]) ;
          END_IF

        C_iSTEP_11 :
         //----------------------------------------------
         // Step 13 : Move down protector
         //----------------------------------------------
          IF NOT(g_bHMP_CmdPhasing)          AND
             NOT(g_bHMP_PhasInProgres)       AND
             ( g_stHMPerfCyc.bTestOn         OR
               NOT(g_stHMPerfCyc.bModTest) ) THEN
            g_stHMPerfCyc.iStep := C_iSTEP_13 ;

            // Action Step 13
            g_stHMPerfCyc.bTestOn := 0 ;

            // Move down protector
            bQ_SOL_HMP_ProtecDown     := 1 ;
            g_stHMPerfCyc.bSynchro_OK := 1 ;
          END_IF

        C_iSTEP_13 :
         //----------------------------------------------
         // Step 14 : Move forward Brush
         //----------------------------------------------
          IF gI_HMP_ProtecDownPE             AND
             ( g_stHMPerfCyc.bTestOn         OR
               NOT(g_stHMPerfCyc.bModTest) ) THEN
            g_stHMPerfCyc.iStep := C_iSTEP_14 ;

            // Action Step 14

            // Move forward Brush
            bQ_SOL_HMP_BrushForward := 1 ;
          END_IF

        C_iSTEP_14 :
         //----------------------------------------------
         // Step 4 : Waiting State
         //----------------------------------------------
          IF NOT(gI_HMP_BrushReturnPE)       AND
             ( g_stHMPerfCyc.bTestOn         OR
               NOT(g_stHMPerfCyc.bModTest) ) THEN
            g_stHMPerfCyc.iStep := C_iSTEP_4 ;

            // Action Step 4
            g_stHMPerfCyc.bTestOn := 0 ;

            // Waiting State
          END_IF

        C_iSTEP_15 :
         //----------------------------------------------
         // Step 16 : Return Brush
         //----------------------------------------------
          IF TRUE                            AND
             ( g_stHMPerfCyc.bTestOn         OR
               NOT(g_stHMPerfCyc.bModTest) ) THEN
            g_stHMPerfCyc.iStep := C_iSTEP_16 ;

            // Action Step 16
            g_stHMPerfCyc.bTestOn := 0 ;

            // Return Brush
            bQ_SOL_HMP_BrushForward := 0 ;
          END_IF

        C_iSTEP_16 :
         //----------------------------------------------
         // Step 17 : Stop Axis
         //           Move up protector
         //----------------------------------------------
          IF gI_HMP_BrushReturnPE            AND
             ( g_stHMPerfCyc.bTestOn         OR
               NOT(g_stHMPerfCyc.bModTest) ) THEN
            g_stHMPerfCyc.iStep := C_iSTEP_17 ;

            // Action Step 17
            g_stHMPerfCyc.bTestOn := 0 ;

            // Stop Axis
            g_stHMPerfCyc.Cmd_Stop      := 1 ;
            gA[15].Cmd_ContinuousMotion := 0 ;
            g_stHMPerfCyc.bSynchro_OK   := 0 ;
            g_stHMPerfCyc.bSlowRot_OK   := 0 ;
            // Move up protector
            bQ_SOL_HMP_ProtecDown := 0 ;
          END_IF

        C_iSTEP_17 :
         //----------------------------------------------
         // Step 18 : Disable Axis
         //----------------------------------------------
          IF NOT(g_stHMPerfCyc.Cmd_Stop)     AND
             gA[15].Ind_StandStill           AND
             NOT(gI_HMP_ProtecDownPE)        AND
             ( g_stHMPerfCyc.bTestOn         OR
               NOT(g_stHMPerfCyc.bModTest) ) THEN
            g_stHMPerfCyc.iStep := C_iSTEP_18 ;

            // Action Step 18
            g_stHMPerfCyc.bTestOn := 0 ;

            g_stHMPerfCyc.Cmd_EnableAxis := 0 ;
          END_IF

        C_iSTEP_18 :
         //----------------------------------------------
         // Step 0 : First step
         //----------------------------------------------
          IF NOT(gA[15].Ind_Enabled)         AND
             NOT(gI_HMP_ProtecDownPE)        AND
             ( g_stHMPerfCyc.bTestOn         OR
               NOT(g_stHMPerfCyc.bModTest) ) THEN
            g_stHMPerfCyc.iStep := C_iSTEP_0 ;

            // Action Step 0
            g_stHMPerfCyc.bTestOn := 0 ;

            g_stHMPerfCyc.bSCyc := 0 ;
            g_stHMPerfCyc.bFCyc := 1 ;
            g_stHMPerfCyc.bCyc  := 0 ;

            g_stHMPerfCyc.bSelProd := NOT(g_stHMPerfCyc.bStopReq) ;
            g_stHMPerfCyc.bStopReq := 0 ;
          END_IF

        END_CASE

END_PROGRAM
```

### Package Logical/BagMachine_Section/BagBundler - A package of related programs and data objects.

### Program Logical/BagMachine_Section/BagBundler/Control
